gfCNCPoint5[21611] = {X 416.6146, Y 101.9777, Z -7.1667, A 0.000, B 0.000, C 0.000 }
gfCNCPoint5[21612] = {X 415.7067, Y 102.0800, Z -7.1667, A 0.000, B 0.000, C 0.000 }
gfCNCPoint5[21613] = {X 396.4059, Y 102.0800, Z -7.1667, A 0.000, B 0.000, C 0.000 }
gfCNCPoint5[21614] = {X 395.4981, Y 101.9777, Z -7.1667, A 0.000, B 0.000, C 0.000 }
gfCNCPoint5[21615] = {X 394.6357, Y 101.6760, Z -7.1667, A 0.000, B 0.000, C 0.000 }
gfCNCPoint5[21616] = {X 393.8621, Y 101.1899, Z -7.1667, A 0.000, B 0.000, C 0.000 }
gfCNCPoint5[21617] = {X 393.2161, Y 100.5438, Z -7.1667, A 0.000, B 0.000, C 0.000 }
gfCNCPoint5[21618] = {X 392.7300, Y 99.7702, Z -7.1667, A 0.000, B 0.000, C 0.000 }
gfCNCPoint5[21619] = {X 392.4282, Y 98.9079, Z -7.1667, A 0.000, B 0.000, C 0.000 }
gfCNCPoint5[21620] = {X 392.3259, Y 98.0000, Z -7.1667, A 0.000, B 0.000, C 0.000 }
gfCNCPoint5[21621] = {X 392.3259, Y 97.0659, Z -7.1667, A 0.000, B 0.000, C 0.000 }
gfCNCPoint5[21622] = {X 392.4280, Y 96.1590, Z -7.1667, A 0.000, B 0.000, C 0.000 }
gfCNCPoint5[21623] = {X 392.7292, Y 95.2974, Z -7.1667, A 0.000, B 0.000, C 0.000 }
gfCNCPoint5[21624] = {X 393.2143, Y 94.5244, Z -7.1667, A 0.000, B 0.000, C 0.000 }
gfCNCPoint5[21625] = {X 393.8591, Y 93.8785, Z -7.1667, A 0.000, B 0.000, C 0.000 }
gfCNCPoint5[21626] = {X 394.6313, Y 93.3921, Z -7.1667, A 0.000, B 0.000, C 0.000 }
gfCNCPoint5[21627] = {X 395.4924, Y 93.0895, Z -7.1667, A 0.000, B 0.000, C 0.000 }
gfCNCPoint5[21628] = {X 396.3991, Y 92.9859, Z -7.1667, A 0.000, B 0.000, C 0.000 }
gfCNCPoint5[21629] = {X 397.3627, Y 92.9425, Z -7.1667, A 0.000, B 0.000, C 0.000 }
gfCNCPoint5[21630] = {X 398.3229, Y 92.8515, Z -7.1667, A 0.000, B 0.000, C 0.000 }
gfCNCPoint5[21631] = {X 399.0264, Y 92.6809, Z -7.1667, A 0.000, B 0.000, C 0.000 }
gfCNCPoint5[21632] = {X 399.6742, Y 92.3580, Z -7.1667, A 0.000, B 0.000, C 0.000 }
gfCNCPoint5[21633] = {X 413.9281, Y 83.2302, Z -7.1667, A 0.000, B 0.000, C 0.000 }
gfCNCPoint5[21634] = {X 411.7658, Y 79.8536, Z -7.1667, A 0.000, B 0.000, C 0.000 }
gfCNCPoint5[21635] = {X 411.7676, Y 79.8524, Z -7.1667, A 0.000, B 0.000, C 0.000 }
gfCNCPoint5[21636] = {X 413.9660, Y 83.2895, Z -7.1667, A 0.000, B 0.000, C 0.000 }
gfCNCPoint5[21637] = {X 428.7544, Y 73.8309, Z -7.1667, A 0.000, B 0.000, C 0.000 }
gfCNCPoint5[21638] = {X 403.8726, Y 64.0690, Z -7.1667, A 0.000, B 0.000, C 0.000 }
gfCNCPoint5[21639] = {X 402.1412, Y 63.4961, Z -7.1667, A 0.000, B 0.000, C 0.000 }
gfCNCPoint5[21640] = {X 400.3574, Y 63.1162, Z -7.1667, A 0.000, B 0.000, C 0.000 }
gfCNCPoint5[21641] = {X 398.5427, Y 62.9340, Z -7.1667, A 0.000, B 0.000, C 0.000 }
gfCNCPoint5[21642] = {X 397.6551, Y 62.8309, Z -7.1667, A 0.000, B 0.000, C 0.000 }
gfCNCPoint5[21643] = {X 396.8125, Y 62.5333, Z -7.1667, A 0.000, B 0.000, C 0.000 }
gfCNCPoint5[21644] = {X 396.0571, Y 62.0560, Z -7.1667, A 0.000, B 0.000, C 0.000 }
gfCNCPoint5[21645] = {X 395.4264, Y 61.4230, Z -7.1667, A 0.000, B 0.000, C 0.000 }
gfCNCPoint5[21646] = {X 394.9520, Y 60.6657, Z -7.1667, A 0.000, B 0.000, C 0.000 }
gfCNCPoint5[21647] = {X 394.6575, Y 59.8221, Z -7.1667, A 0.000, B 0.000, C 0.000 }
gfCNCPoint5[21648] = {X 394.5577, Y 58.9341, Z -7.1667, A 0.000, B 0.000, C 0.000 }
gfCNCPoint5[21649] = {X 394.5577, Y 58.0000, Z -7.1667, A 0.000, B 0.000, C 0.000 }
gfCNCPoint5[21650] = {X 394.6580, Y 57.1099, Z -7.1667, A 0.000, B 0.000, C 0.000 }
gfCNCPoint5[21651] = {X 394.9538, Y 56.2645, Z -7.1667, A 0.000, B 0.000, C 0.000 }
gfCNCPoint5[21652] = {X 395.4304, Y 55.5060, Z -7.1667, A 0.000, B 0.000, C 0.000 }
gfCNCPoint5[21653] = {X 396.0638, Y 54.8727, Z -7.1667, A 0.000, B 0.000, C 0.000 }
gfCNCPoint5[21654] = {X 396.8222, Y 54.3961, Z -7.1667, A 0.000, B 0.000, C 0.000 }
gfCNCPoint5[21655] = {X 397.6676, Y 54.1003, Z -7.1667, A 0.000, B 0.000, C 0.000 }
gfCNCPoint5[21656] = {X 398.5577, Y 54.0000, Z -7.1667, A 0.000, B 0.000, C 0.000 }
gfCNCPoint5[21657] = {X 419.4886, Y 54.0000, Z -7.1667, A 0.000, B 0.000, C 0.000 }
gfCNCPoint5[21658] = {X 420.3787, Y 54.1003, Z -7.1667, A 0.000, B 0.000, C 0.000 }
gfCNCPoint5[21659] = {X 421.2241, Y 54.3961, Z -7.1667, A 0.000, B 0.000, C 0.000 }
gfCNCPoint5[21660] = {X 421.9826, Y 54.8727, Z -7.1667, A 0.000, B 0.000, C 0.000 }
gfCNCPoint5[21661] = {X 422.6159, Y 55.5060, Z -7.1667, A 0.000, B 0.000, C 0.000 }
gfCNCPoint5[21662] = {X 423.0925, Y 56.2645, Z -7.1667, A 0.000, B 0.000, C 0.000 }
gfCNCPoint5[21663] = {X 423.3883, Y 57.1099, Z -7.1667, A 0.000, B 0.000, C 0.000 }
gfCNCPoint5[21664] = {X 423.4886, Y 58.0000, Z -7.1667, A 0.000, B 0.000, C 0.000 }
gfCNCPoint5[21665] = {X 423.4886, Y 58.4503, Z -7.1667, A 0.000, B 0.000, C 0.000 }
gfCNCPoint5[21666] = {X 429.4945, Y 60.7902, Z -7.1667, A 0.000, B 0.000, C 0.000 }
gfCNCPoint5[21667] = {X 458.1780, Y 72.1710, Z -7.1667, A 0.000, B 0.000, C 0.000 }
gfCNCPoint5[21668] = {X 458.1783, Y 63.0394, Z -7.1667, A 0.000, B 0.000, C 0.000 }
gfCNCPoint5[21669] = {X 458.1841, Y 62.9246, Z -7.1667, A 0.000, B 0.000, C 0.000 }
gfCNCPoint5[21670] = {X 458.0117, Y 62.9089, Z -7.1667, A 0.000, B 0.000, C 0.000 }
gfCNCPoint5[21671] = {X 457.8402, Y 62.8858, Z -7.1667, A 0.000, B 0.000, C 0.000 }
gfCNCPoint5[21672] = {X 456.9338, Y 62.6316, Z -7.1667, A 0.000, B 0.000, C 0.000 }
gfCNCPoint5[21673] = {X 456.1119, Y 62.1727, Z -7.1667, A 0.000, B 0.000, C 0.000 }
gfCNCPoint5[21674] = {X 455.4201, Y 61.5343, Z -7.1667, A 0.000, B 0.000, C 0.000 }
gfCNCPoint5[21675] = {X 454.8966, Y 60.7519, Z -7.1667, A 0.000, B 0.000, C 0.000 }
gfCNCPoint5[21676] = {X 454.5704, Y 59.8689, Z -7.1667, A 0.000, B 0.000, C 0.000 }
gfCNCPoint5[21677] = {X 454.4596, Y 58.9341, Z -7.1667, A 0.000, B 0.000, C 0.000 }
gfCNCPoint5[21678] = {X 454.4596, Y 58.0000, Z -7.1667, A 0.000, B 0.000, C 0.000 }
gfCNCPoint5[21679] = {X 454.5599, Y 57.1099, Z -7.1667, A 0.000, B 0.000, C 0.000 }
gfCNCPoint5[21680] = {X 454.8557, Y 56.2645, Z -7.1667, A 0.000, B 0.000, C 0.000 }
gfCNCPoint5[21681] = {X 455.3323, Y 55.5060, Z -7.1667, A 0.000, B 0.000, C 0.000 }
gfCNCPoint5[21682] = {X 455.9656, Y 54.8727, Z -7.1667, A 0.000, B 0.000, C 0.000 }
gfCNCPoint5[21683] = {X 456.7241, Y 54.3961, Z -7.1667, A 0.000, B 0.000, C 0.000 }
gfCNCPoint5[21684] = {X 457.5695, Y 54.1003, Z -7.1667, A 0.000, B 0.000, C 0.000 }
gfCNCPoint5[21685] = {X 458.4596, Y 54.0000, Z -7.1667, A 0.000, B 0.000, C 0.000 }
gfCNCPoint5[21686] = {X 475.0000, Y 54.0000, Z -7.1667, A 0.000, B 0.000, C 0.000 }
gfCNCPoint5[21687] = {X 475.8901, Y 54.1003, Z -7.1667, A 0.000, B 0.000, C 0.000 }
gfCNCPoint5[21688] = {X 476.7355, Y 54.3961, Z -7.1667, A 0.000, B 0.000, C 0.000 }
gfCNCPoint5[21689] = {X 477.4940, Y 54.8727, Z -7.1667, A 0.000, B 0.000, C 0.000 }
gfCNCPoint5[21690] = {X 478.1273, Y 55.5060, Z -7.1667, A 0.000, B 0.000, C 0.000 }
gfCNCPoint5[21691] = {X 478.6039, Y 56.2645, Z -7.1667, A 0.000, B 0.000, C 0.000 }
gfCNCPoint5[21692] = {X 478.8997, Y 57.1099, Z -7.1667, A 0.000, B 0.000, C 0.000 }
gfCNCPoint5[21693] = {X 479.0000, Y 58.0000, Z -7.1667, A 0.000, B 0.000, C 0.000 }
gfCNCPoint5[21694] = {X 478.9999, Y 58.9671, Z -7.1667, A 0.000, B 0.000, C 0.000 }
gfCNCPoint5[21695] = {X 478.8827, Y 59.8957, Z -7.1667, A 0.000, B 0.000, C 0.000 }
gfCNCPoint5[21696] = {X 478.5529, Y 60.7716, Z -7.1667, A 0.000, B 0.000, C 0.000 }
gfCNCPoint5[21697] = {X 478.0287, Y 61.5469, Z -7.1667, A 0.000, B 0.000, C 0.000 }
gfCNCPoint5[21698] = {X 477.3386, Y 62.1792, Z -7.1667, A 0.000, B 0.000, C 0.000 }
gfCNCPoint5[21699] = {X 476.5204, Y 62.6338, Z -7.1667, A 0.000, B 0.000, C 0.000 }
gfCNCPoint5[21700] = {X 475.6191, Y 62.8859, Z -7.1667, A 0.000, B 0.000, C 0.000 }
gfCNCPoint5[21701] = {X 475.4521, Y 62.9084, Z -7.1667, A 0.000, B 0.000, C 0.000 }
gfCNCPoint5[21702] = {X 475.2843, Y 62.9240, Z -7.1667, A 0.000, B 0.000, C 0.000 }
gfCNCPoint5[21703] = {X 475.2810, Y 63.2811, Z -7.1667, A 0.000, B 0.000, C 0.000 }
gfCNCPoint5[21704] = {X 475.2814, Y 93.0285, Z -7.1667, A 0.000, B 0.000, C 0.000 }
gfCNCPoint5[21705] = {X 475.7846, Y 93.1405, Z -7.1667, A 0.000, B 0.000, C 0.000 }
gfCNCPoint5[21706] = {X 476.2789, Y 93.2866, Z -7.1667, A 0.000, B 0.000, C 0.000 }
gfCNCPoint5[21707] = {X 477.0319, Y 93.6280, Z -7.1667, A 0.000, B 0.000, C 0.000 }
gfCNCPoint5[21708] = {X 477.6982, Y 94.1177, Z -7.1667, A 0.000, B 0.000, C 0.000 }
gfCNCPoint5[21709] = {X 478.2488, Y 94.7346, Z -7.1667, A 0.000, B 0.000, C 0.000 }
gfCNCPoint5[21710] = {X 478.6600, Y 95.4519, Z -7.1667, A 0.000, B 0.000, C 0.000 }
gfCNCPoint5[21711] = {X 478.9141, Y 96.2388, Z -7.1667, A 0.000, B 0.000, C 0.000 }
gfCNCPoint5[21712] = {X 479.0000, Y 97.0611, Z -7.1667, A 0.000, B 0.000, C 0.000 }
gfCNCPoint5[21713] = {X 479.0000, Y 98.0000, Z -7.1667, A 0.000, B 0.000, C 0.000 }
gfCNCPoint5[21714] = {X 478.8997, Y 98.8901, Z -7.1667, A 0.000, B 0.000, C 0.000 }
gfCNCPoint5[21715] = {X 478.6039, Y 99.7355, Z -7.1667, A 0.000, B 0.000, C 0.000 }
gfCNCPoint5[21716] = {X 478.1273, Y 100.4940, Z -7.1667, A 0.000, B 0.000, C 0.000 }
gfCNCPoint5[21717] = {X 477.4940, Y 101.1273, Z -7.1667, A 0.000, B 0.000, C 0.000 }
gfCNCPoint5[21718] = {X 476.7355, Y 101.6039, Z -7.1667, A 0.000, B 0.000, C 0.000 }
gfCNCPoint5[21719] = {X 475.8901, Y 101.8997, Z -7.1667, A 0.000, B 0.000, C 0.000 }
gfCNCPoint5[21720] = {X 475.0000, Y 102.0000, Z -7.1667, A 0.000, B 0.000, C 0.000 }
gfCNCPoint5[21721] = {X 458.4596, Y 102.0000, Z -7.1667, A 0.000, B 0.000, C 0.000 }
gfCNCPoint5[21722] = {X 457.5695, Y 101.8997, Z -7.1667, A 0.000, B 0.000, C 0.000 }
gfCNCPoint5[21723] = {X 456.7241, Y 101.6039, Z -7.1667, A 0.000, B 0.000, C 0.000 }
gfCNCPoint5[21724] = {X 455.9656, Y 101.1273, Z -7.1667, A 0.000, B 0.000, C 0.000 }
gfCNCPoint5[21725] = {X 455.3323, Y 100.4940, Z -7.1667, A 0.000, B 0.000, C 0.000 }
gfCNCPoint5[21726] = {X 454.8557, Y 99.7355, Z -7.1667, A 0.000, B 0.000, C 0.000 }
gfCNCPoint5[21727] = {X 454.5599, Y 98.8901, Z -7.1667, A 0.000, B 0.000, C 0.000 }
gfCNCPoint5[21728] = {X 454.4596, Y 98.0000, Z -7.1667, A 0.000, B 0.000, C 0.000 }
gfCNCPoint5[21729] = {X 454.4596, Y 97.0659, Z -7.1667, A 0.000, B 0.000, C 0.000 }
gfCNCPoint5[21730] = {X 454.5511, Y 96.2154, Z -7.1667, A 0.000, B 0.000, C 0.000 }
gfCNCPoint5[21731] = {X 454.8213, Y 95.4037, Z -7.1667, A 0.000, B 0.000, C 0.000 }
gfCNCPoint5[21732] = {X 455.2580, Y 94.6681, Z -7.1667, A 0.000, B 0.000, C 0.000 }
gfCNCPoint5[21733] = {X 455.8411, Y 94.0422, Z -7.1667, A 0.000, B 0.000, C 0.000 }
gfCNCPoint5[21734] = {X 456.5439, Y 93.5545, Z -7.1667, A 0.000, B 0.000, C 0.000 }
gfCNCPoint5[21735] = {X 457.3344, Y 93.2275, Z -7.1667, A 0.000, B 0.000, C 0.000 }
gfCNCPoint5[21736] = {X 458.1763, Y 93.0760, Z -7.1667, A 0.000, B 0.000, C 0.000 }
gfCNCPoint5[21737] = {X 458.1763, Y 85.3767, Z -7.1667, A 0.000, B 0.000, C 0.000 }
gfCNCPoint5[21738] = {X 445.0152, Y 80.2175, Z -7.1667, A 0.000, B 0.000, C 0.000 }
gfCNCPoint5[21739] = {X 444.8242, Y 80.1425, Z -7.1667, A 0.000, B 0.000, C 0.000 }
gfCNCPoint5[21740] = {X 419.7033, Y 96.4151, Z -7.1667, A 0.000, B 0.000, C 0.000 }
gfCNCPoint5[21741] = {X 419.7067, Y 97.0659, Z -7.1667, A 0.000, B 0.000, C 0.000 }
gfCNCPoint5[21742] = {X 419.7067, Y 98.0000, Z -7.1667, A 0.000, B 0.000, C 0.000 }
gfCNCPoint5[21743] = {X 419.6064, Y 98.8901, Z -7.1667, A 0.000, B 0.000, C 0.000 }
gfCNCPoint5[21744] = {X 419.3106, Y 99.7355, Z -7.1667, A 0.000, B 0.000, C 0.000 }
gfCNCPoint5[21745] = {X 418.8340, Y 100.4940, Z -7.1667, A 0.000, B 0.000, C 0.000 }
gfCNCPoint5[21746] = {X 418.2007, Y 101.1273, Z -7.1667, A 0.000, B 0.000, C 0.000 }
gfCNCPoint5[21747] = {X 417.4422, Y 101.6039, Z -7.1667, A 0.000, B 0.000, C 0.000 }
gfCNCPoint5[21748] = {X 416.5968, Y 101.8997, Z -7.1667, A 0.000, B 0.000, C 0.000 }
gfCNCPoint5[21749] = {X 415.7067, Y 102.0000, Z -7.1667, A 0.000, B 0.000, C 0.000 }
gfCNCPoint5[21750] = {X 396.4059, Y 102.0000, Z -7.1667, A 0.000, B 0.000, C 0.000 }
gfCNCPoint5[21751] = {X 395.5159, Y 101.8997, Z -7.1667, A 0.000, B 0.000, C 0.000 }
gfCNCPoint5[21752] = {X 394.6704, Y 101.6039, Z -7.1667, A 0.000, B 0.000, C 0.000 }
gfCNCPoint5[21753] = {X 393.9120, Y 101.1273, Z -7.1667, A 0.000, B 0.000, C 0.000 }
gfCNCPoint5[21754] = {X 393.2786, Y 100.4940, Z -7.1667, A 0.000, B 0.000, C 0.000 }
gfCNCPoint5[21755] = {X 392.8021, Y 99.7355, Z -7.1667, A 0.000, B 0.000, C 0.000 }
gfCNCPoint5[21756] = {X 392.5062, Y 98.8901, Z -7.1667, A 0.000, B 0.000, C 0.000 }
gfCNCPoint5[21757] = {X 392.4059, Y 98.0000, Z -7.1667, A 0.000, B 0.000, C 0.000 }
gfCNCPoint5[21758] = {X 392.4059, Y 97.0659, Z -7.1667, A 0.000, B 0.000, C 0.000 }
gfCNCPoint5[21759] = {X 392.5060, Y 96.1767, Z -7.1667, A 0.000, B 0.000, C 0.000 }
gfCNCPoint5[21760] = {X 392.8013, Y 95.3319, Z -7.1667, A 0.000, B 0.000, C 0.000 }
gfCNCPoint5[21761] = {X 393.2770, Y 94.5740, Z -7.1667, A 0.000, B 0.000, C 0.000 }
gfCNCPoint5[21762] = {X 393.9093, Y 93.9407, Z -7.1667, A 0.000, B 0.000, C 0.000 }
gfCNCPoint5[21763] = {X 394.6666, Y 93.4639, Z -7.1667, A 0.000, B 0.000, C 0.000 }
gfCNCPoint5[21764] = {X 395.5109, Y 93.1674, Z -7.1667, A 0.000, B 0.000, C 0.000 }
gfCNCPoint5[21765] = {X 396.4000, Y 93.0659, Z -7.1667, A 0.000, B 0.000, C 0.000 }
gfCNCPoint5[21766] = {X 397.3680, Y 93.0223, Z -7.1667, A 0.000, B 0.000, C 0.000 }
gfCNCPoint5[21767] = {X 398.3327, Y 92.9309, Z -7.1667, A 0.000, B 0.000, C 0.000 }
gfCNCPoint5[21768] = {X 399.0537, Y 92.7561, Z -7.1667, A 0.000, B 0.000, C 0.000 }
gfCNCPoint5[21769] = {X 399.7177, Y 92.4252, Z -7.1667, A 0.000, B 0.000, C 0.000 }
gfCNCPoint5[21770] = {X 404.3153, Y 89.4621, Z -7.1667, A 0.000, B 0.000, C 0.000 }
gfCNCPoint5[21771] = {X 413.9660, Y 83.2895, Z -7.1667, A 0.000, B 0.000, C 0.000 }
gfCNCPoint5[21772] = {X 411.7676, Y 79.8524, Z -7.1667, A 0.000, B 0.000, C 0.000 }
gfCNCPoint5[21773] = {X 411.7676, Y 79.8524, Z -4.1667, A 0.000, B 0.000, C 0.000 }
gfCNCPoint5[21774] = {X 411.7676, Y 79.8524, Z 11.0000, A 0.000, B 0.000, C 0.000 }
gfCNCPoint5[21775] = {X 466.3117, Y 28.5934, Z 11.0000, A 0.000, B 0.000, C 0.000 }
gfCNCPoint5[21776] = {X 466.3117, Y 28.5934, Z -4.1667, A 0.000, B 0.000, C 0.000 }
gfCNCPoint5[21777] = {X 466.3117, Y 28.5934, Z -7.1667, A 0.000, B 0.000, C 0.000 }
gfCNCPoint5[21778] = {X 462.2317, Y 28.5935, Z -7.1667, A 0.000, B 0.000, C 0.000 }
gfCNCPoint5[21779] = {X 462.2320, Y 40.9142, Z -7.1667, A 0.000, B 0.000, C 0.000 }
gfCNCPoint5[21780] = {X 462.2403, Y 40.9211, Z -7.1667, A 0.000, B 0.000, C 0.000 }
gfCNCPoint5[21781] = {X 462.8748, Y 41.5915, Z -7.1667, A 0.000, B 0.000, C 0.000 }
gfCNCPoint5[21782] = {X 463.3524, Y 42.3815, Z -7.1667, A 0.000, B 0.000, C 0.000 }
gfCNCPoint5[21783] = {X 463.6513, Y 43.2548, Z -7.1667, A 0.000, B 0.000, C 0.000 }
gfCNCPoint5[21784] = {X 463.7578, Y 44.1718, Z -7.1667, A 0.000, B 0.000, C 0.000 }
gfCNCPoint5[21785] = {X 463.7579, Y 45.0000, Z -7.1667, A 0.000, B 0.000, C 0.000 }
gfCNCPoint5[21786] = {X 463.6496, Y 45.9613, Z -7.1667, A 0.000, B 0.000, C 0.000 }
gfCNCPoint5[21787] = {X 463.3301, Y 46.8744, Z -7.1667, A 0.000, B 0.000, C 0.000 }
gfCNCPoint5[21788] = {X 462.8155, Y 47.6935, Z -7.1667, A 0.000, B 0.000, C 0.000 }
gfCNCPoint5[21789] = {X 462.1314, Y 48.3775, Z -7.1667, A 0.000, B 0.000, C 0.000 }
gfCNCPoint5[21790] = {X 461.3123, Y 48.8922, Z -7.1667, A 0.000, B 0.000, C 0.000 }
gfCNCPoint5[21791] = {X 460.3992, Y 49.2117, Z -7.1667, A 0.000, B 0.000, C 0.000 }
gfCNCPoint5[21792] = {X 459.4379, Y 49.3200, Z -7.1667, A 0.000, B 0.000, C 0.000 }
gfCNCPoint5[21793] = {X 452.9945, Y 49.3200, Z -7.1667, A 0.000, B 0.000, C 0.000 }
gfCNCPoint5[21794] = {X 452.0380, Y 49.2128, Z -7.1667, A 0.000, B 0.000, C 0.000 }
gfCNCPoint5[21795] = {X 451.1291, Y 48.8965, Z -7.1667, A 0.000, B 0.000, C 0.000 }
gfCNCPoint5[21796] = {X 450.3127, Y 48.3868, Z -7.1667, A 0.000, B 0.000, C 0.000 }
gfCNCPoint5[21797] = {X 449.6294, Y 47.7091, Z -7.1667, A 0.000, B 0.000, C 0.000 }
gfCNCPoint5[21798] = {X 449.1132, Y 46.8968, Z -7.1667, A 0.000, B 0.000, C 0.000 }
gfCNCPoint5[21799] = {X 448.7895, Y 45.9905, Z -7.1667, A 0.000, B 0.000, C 0.000 }
gfCNCPoint5[21800] = {X 448.6746, Y 45.0349, Z -7.1667, A 0.000, B 0.000, C 0.000 }
gfCNCPoint5[21801] = {X 448.6749, Y 44.1494, Z -7.1667, A 0.000, B 0.000, C 0.000 }
gfCNCPoint5[21802] = {X 448.7853, Y 43.2364, Z -7.1667, A 0.000, B 0.000, C 0.000 }
gfCNCPoint5[21803] = {X 449.0865, Y 42.3675, Z -7.1667, A 0.000, B 0.000, C 0.000 }
gfCNCPoint5[21804] = {X 449.5648, Y 41.5821, Z -7.1667, A 0.000, B 0.000, C 0.000 }
gfCNCPoint5[21805] = {X 450.1984, Y 40.9157, Z -7.1667, A 0.000, B 0.000, C 0.000 }
gfCNCPoint5[21806] = {X 450.1984, Y 34.4738, Z -7.1667, A 0.000, B 0.000, C 0.000 }
gfCNCPoint5[21807] = {X 447.4755, Y 34.4738, Z -7.1667, A 0.000, B 0.000, C 0.000 }
gfCNCPoint5[21808] = {X 443.1901, Y 42.8178, Z -7.1667, A 0.000, B 0.000, C 0.000 }
gfCNCPoint5[21809] = {X 443.1949, Y 42.8312, Z -7.1667, A 0.000, B 0.000, C 0.000 }
gfCNCPoint5[21810] = {X 443.3606, Y 43.4918, Z -7.1667, A 0.000, B 0.000, C 0.000 }
gfCNCPoint5[21811] = {X 443.4203, Y 44.1703, Z -7.1667, A 0.000, B 0.000, C 0.000 }
gfCNCPoint5[21812] = {X 443.4205, Y 45.0000, Z -7.1667, A 0.000, B 0.000, C 0.000 }
gfCNCPoint5[21813] = {X 443.3122, Y 45.9613, Z -7.1667, A 0.000, B 0.000, C 0.000 }
gfCNCPoint5[21814] = {X 442.9927, Y 46.8744, Z -7.1667, A 0.000, B 0.000, C 0.000 }
gfCNCPoint5[21815] = {X 442.4780, Y 47.6935, Z -7.1667, A 0.000, B 0.000, C 0.000 }
gfCNCPoint5[21816] = {X 441.7939, Y 48.3775, Z -7.1667, A 0.000, B 0.000, C 0.000 }
gfCNCPoint5[21817] = {X 440.9748, Y 48.8922, Z -7.1667, A 0.000, B 0.000, C 0.000 }
gfCNCPoint5[21818] = {X 440.0618, Y 49.2117, Z -7.1667, A 0.000, B 0.000, C 0.000 }
gfCNCPoint5[21819] = {X 439.1005, Y 49.3200, Z -7.1667, A 0.000, B 0.000, C 0.000 }
gfCNCPoint5[21820] = {X 432.5144, Y 49.3200, Z -7.1667, A 0.000, B 0.000, C 0.000 }
gfCNCPoint5[21821] = {X 431.5531, Y 49.2117, Z -7.1667, A 0.000, B 0.000, C 0.000 }
gfCNCPoint5[21822] = {X 430.6401, Y 48.8922, Z -7.1667, A 0.000, B 0.000, C 0.000 }
gfCNCPoint5[21823] = {X 429.8210, Y 48.3775, Z -7.1667, A 0.000, B 0.000, C 0.000 }
gfCNCPoint5[21824] = {X 429.1369, Y 47.6935, Z -7.1667, A 0.000, B 0.000, C 0.000 }
gfCNCPoint5[21825] = {X 428.6223, Y 46.8745, Z -7.1667, A 0.000, B 0.000, C 0.000 }
gfCNCPoint5[21826] = {X 428.3027, Y 45.9614, Z -7.1667, A 0.000, B 0.000, C 0.000 }
gfCNCPoint5[21827] = {X 428.1944, Y 45.0001, Z -7.1667, A 0.000, B 0.000, C 0.000 }
gfCNCPoint5[21828] = {X 428.1948, Y 44.1494, Z -7.1667, A 0.000, B 0.000, C 0.000 }
gfCNCPoint5[21829] = {X 428.2925, Y 43.2935, Z -7.1667, A 0.000, B 0.000, C 0.000 }
gfCNCPoint5[21830] = {X 428.5580, Y 42.4740, Z -7.1667, A 0.000, B 0.000, C 0.000 }
gfCNCPoint5[21831] = {X 428.9809, Y 41.7236, Z -7.1667, A 0.000, B 0.000, C 0.000 }
gfCNCPoint5[21832] = {X 429.5442, Y 41.0719, Z -7.1667, A 0.000, B 0.000, C 0.000 }
gfCNCPoint5[21833] = {X 430.2256, Y 40.5449, Z -7.1667, A 0.000, B 0.000, C 0.000 }
gfCNCPoint5[21834] = {X 430.9981, Y 40.1637, Z -7.1667, A 0.000, B 0.000, C 0.000 }
gfCNCPoint5[21835] = {X 434.9867, Y 32.3563, Z -7.1667, A 0.000, B 0.000, C 0.000 }
gfCNCPoint5[21836] = {X 433.8226, Y 31.5747, Z -7.1667, A 0.000, B 0.000, C 0.000 }
gfCNCPoint5[21837] = {X 432.7640, Y 30.6552, Z -7.1667, A 0.000, B 0.000, C 0.000 }
gfCNCPoint5[21838] = {X 431.8273, Y 29.6119, Z -7.1667, A 0.000, B 0.000, C 0.000 }
gfCNCPoint5[21839] = {X 431.0267, Y 28.4607, Z -7.1667, A 0.000, B 0.000, C 0.000 }
gfCNCPoint5[21840] = {X 430.3746, Y 27.2194, Z -7.1667, A 0.000, B 0.000, C 0.000 }
gfCNCPoint5[21841] = {X 429.8811, Y 25.9069, Z -7.1667, A 0.000, B 0.000, C 0.000 }
gfCNCPoint5[21842] = {X 429.4497, Y 24.0606, Z -7.1667, A 0.000, B 0.000, C 0.000 }
gfCNCPoint5[21843] = {X 429.2325, Y 22.1770, Z -7.1667, A 0.000, B 0.000, C 0.000 }
gfCNCPoint5[21844] = {X 429.2323, Y 20.2810, Z -7.1667, A 0.000, B 0.000, C 0.000 }
gfCNCPoint5[21845] = {X 429.4491, Y 18.3974, Z -7.1667, A 0.000, B 0.000, C 0.000 }
gfCNCPoint5[21846] = {X 429.8800, Y 16.5509, Z -7.1667, A 0.000, B 0.000, C 0.000 }
gfCNCPoint5[21847] = {X 430.4498, Y 15.0197, Z -7.1667, A 0.000, B 0.000, C 0.000 }
gfCNCPoint5[21848] = {X 431.2251, Y 13.5816, Z -7.1667, A 0.000, B 0.000, C 0.000 }
gfCNCPoint5[21849] = {X 432.1911, Y 12.2641, Z -7.1667, A 0.000, B 0.000, C 0.000 }
gfCNCPoint5[21850] = {X 433.3295, Y 11.0922, Z -7.1667, A 0.000, B 0.000, C 0.000 }
gfCNCPoint5[21851] = {X 434.6185, Y 10.0883, Z -7.1667, A 0.000, B 0.000, C 0.000 }
gfCNCPoint5[21852] = {X 436.0334, Y 9.2716, Z -7.1667, A 0.000, B 0.000, C 0.000 }
gfCNCPoint5[21853] = {X 437.5474, Y 8.6577, Z -7.1667, A 0.000, B 0.000, C 0.000 }
gfCNCPoint5[21854] = {X 439.1316, Y 8.2581, Z -7.1667, A 0.000, B 0.000, C 0.000 }
gfCNCPoint5[21855] = {X 441.2286, Y 7.9678, Z -7.1667, A 0.000, B 0.000, C 0.000 }
gfCNCPoint5[21856] = {X 443.3436, Y 7.8736, Z -7.1667, A 0.000, B 0.000, C 0.000 }
gfCNCPoint5[21857] = {X 444.0357, Y 7.8696, Z -7.1667, A 0.000, B 0.000, C 0.000 }
gfCNCPoint5[21858] = {X 459.4469, Y 7.8696, Z -7.1667, A 0.000, B 0.000, C 0.000 }
gfCNCPoint5[21859] = {X 460.4062, Y 7.9777, Z -7.1667, A 0.000, B 0.000, C 0.000 }
gfCNCPoint5[21860] = {X 461.3174, Y 8.2965, Z -7.1667, A 0.000, B 0.000, C 0.000 }
gfCNCPoint5[21861] = {X 462.1348, Y 8.8101, Z -7.1667, A 0.000, B 0.000, C 0.000 }
gfCNCPoint5[21862] = {X 462.8174, Y 9.4927, Z -7.1667, A 0.000, B 0.000, C 0.000 }
gfCNCPoint5[21863] = {X 463.3310, Y 10.3101, Z -7.1667, A 0.000, B 0.000, C 0.000 }
gfCNCPoint5[21864] = {X 463.6499, Y 11.2213, Z -7.1667, A 0.000, B 0.000, C 0.000 }
gfCNCPoint5[21865] = {X 463.7579, Y 12.1806, Z -7.1667, A 0.000, B 0.000, C 0.000 }
gfCNCPoint5[21866] = {X 463.7579, Y 12.9782, Z -7.1667, A 0.000, B 0.000, C 0.000 }
gfCNCPoint5[21867] = {X 463.6566, Y 13.9077, Z -7.1667, A 0.000, B 0.000, C 0.000 }
gfCNCPoint5[21868] = {X 463.3577, Y 14.7936, Z -7.1667, A 0.000, B 0.000, C 0.000 }
gfCNCPoint5[21869] = {X 462.8751, Y 15.5945, Z -7.1667, A 0.000, B 0.000, C 0.000 }
gfCNCPoint5[21870] = {X 462.2315, Y 16.2728, Z -7.1667, A 0.000, B 0.000, C 0.000 }
gfCNCPoint5[21871] = {X 462.2317, Y 28.5935, Z -7.1667, A 0.000, B 0.000, C 0.000 }
gfCNCPoint5[21872] = {X 466.2317, Y 28.5934, Z -7.1667, A 0.000, B 0.000, C 0.000 }
gfCNCPoint5[21873] = {X 462.1517, Y 28.5935, Z -7.1667, A 0.000, B 0.000, C 0.000 }
gfCNCPoint5[21874] = {X 462.1520, Y 40.9519, Z -7.1667, A 0.000, B 0.000, C 0.000 }
gfCNCPoint5[21875] = {X 462.1889, Y 40.9824, Z -7.1667, A 0.000, B 0.000, C 0.000 }
gfCNCPoint5[21876] = {X 462.8115, Y 41.6404, Z -7.1667, A 0.000, B 0.000, C 0.000 }
gfCNCPoint5[21877] = {X 463.2801, Y 42.4156, Z -7.1667, A 0.000, B 0.000, C 0.000 }
gfCNCPoint5[21878] = {X 463.5733, Y 43.2726, Z -7.1667, A 0.000, B 0.000, C 0.000 }
gfCNCPoint5[21879] = {X 463.6778, Y 44.1724, Z -7.1667, A 0.000, B 0.000, C 0.000 }
gfCNCPoint5[21880] = {X 463.6779, Y 45.0000, Z -7.1667, A 0.000, B 0.000, C 0.000 }
gfCNCPoint5[21881] = {X 463.5716, Y 45.9435, Z -7.1667, A 0.000, B 0.000, C 0.000 }
gfCNCPoint5[21882] = {X 463.2580, Y 46.8397, Z -7.1667, A 0.000, B 0.000, C 0.000 }
gfCNCPoint5[21883] = {X 462.7529, Y 47.6436, Z -7.1667, A 0.000, B 0.000, C 0.000 }
gfCNCPoint5[21884] = {X 462.0815, Y 48.3150, Z -7.1667, A 0.000, B 0.000, C 0.000 }
gfCNCPoint5[21885] = {X 461.2776, Y 48.8201, Z -7.1667, A 0.000, B 0.000, C 0.000 }
gfCNCPoint5[21886] = {X 460.3814, Y 49.1337, Z -7.1667, A 0.000, B 0.000, C 0.000 }
gfCNCPoint5[21887] = {X 459.4379, Y 49.2400, Z -7.1667, A 0.000, B 0.000, C 0.000 }
gfCNCPoint5[21888] = {X 452.9945, Y 49.2400, Z -7.1667, A 0.000, B 0.000, C 0.000 }
gfCNCPoint5[21889] = {X 452.0558, Y 49.1348, Z -7.1667, A 0.000, B 0.000, C 0.000 }
gfCNCPoint5[21890] = {X 451.1636, Y 48.8243, Z -7.1667, A 0.000, B 0.000, C 0.000 }
gfCNCPoint5[21891] = {X 450.3624, Y 48.3241, Z -7.1667, A 0.000, B 0.000, C 0.000 }
gfCNCPoint5[21892] = {X 449.6918, Y 47.6589, Z -7.1667, A 0.000, B 0.000, C 0.000 }
gfCNCPoint5[21893] = {X 449.1851, Y 46.8617, Z -7.1667, A 0.000, B 0.000, C 0.000 }
gfCNCPoint5[21894] = {X 448.8674, Y 45.9721, Z -7.1667, A 0.000, B 0.000, C 0.000 }
gfCNCPoint5[21895] = {X 448.7546, Y 45.0343, Z -7.1667, A 0.000, B 0.000, C 0.000 }
gfCNCPoint5[21896] = {X 448.7549, Y 44.1505, Z -7.1667, A 0.000, B 0.000, C 0.000 }
gfCNCPoint5[21897] = {X 448.8654, Y 43.2454, Z -7.1667, A 0.000, B 0.000, C 0.000 }
gfCNCPoint5[21898] = {X 449.1668, Y 42.3850, Z -7.1667, A 0.000, B 0.000, C 0.000 }
gfCNCPoint5[21899] = {X 449.6452, Y 41.6088, Z -7.1667, A 0.000, B 0.000, C 0.000 }
gfCNCPoint5[21900] = {X 450.2784, Y 40.9529, Z -7.1667, A 0.000, B 0.000, C 0.000 }
gfCNCPoint5[21901] = {X 450.2784, Y 34.3938, Z -7.1667, A 0.000, B 0.000, C 0.000 }
gfCNCPoint5[21902] = {X 447.4266, Y 34.3938, Z -7.1667, A 0.000, B 0.000, C 0.000 }
gfCNCPoint5[21903] = {X 443.1031, Y 42.8122, Z -7.1667, A 0.000, B 0.000, C 0.000 }
gfCNCPoint5[21904] = {X 443.1194, Y 42.8575, Z -7.1667, A 0.000, B 0.000, C 0.000 }
gfCNCPoint5[21905] = {X 443.2817, Y 43.5055, Z -7.1667, A 0.000, B 0.000, C 0.000 }
gfCNCPoint5[21906] = {X 443.3403, Y 44.1710, Z -7.1667, A 0.000, B 0.000, C 0.000 }
gfCNCPoint5[21907] = {X 443.3405, Y 45.0000, Z -7.1667, A 0.000, B 0.000, C 0.000 }
gfCNCPoint5[21908] = {X 443.2342, Y 45.9435, Z -7.1667, A 0.000, B 0.000, C 0.000 }
gfCNCPoint5[21909] = {X 442.9206, Y 46.8397, Z -7.1667, A 0.000, B 0.000, C 0.000 }
gfCNCPoint5[21910] = {X 442.4154, Y 47.6436, Z -7.1667, A 0.000, B 0.000, C 0.000 }
gfCNCPoint5[21911] = {X 441.7441, Y 48.3150, Z -7.1667, A 0.000, B 0.000, C 0.000 }
gfCNCPoint5[21912] = {X 440.9401, Y 48.8201, Z -7.1667, A 0.000, B 0.000, C 0.000 }
gfCNCPoint5[21913] = {X 440.0440, Y 49.1337, Z -7.1667, A 0.000, B 0.000, C 0.000 }
gfCNCPoint5[21914] = {X 439.1005, Y 49.2400, Z -7.1667, A 0.000, B 0.000, C 0.000 }
gfCNCPoint5[21915] = {X 432.5144, Y 49.2400, Z -7.1667, A 0.000, B 0.000, C 0.000 }
gfCNCPoint5[21916] = {X 431.5709, Y 49.1337, Z -7.1667, A 0.000, B 0.000, C 0.000 }
gfCNCPoint5[21917] = {X 430.6748, Y 48.8201, Z -7.1667, A 0.000, B 0.000, C 0.000 }
gfCNCPoint5[21918] = {X 429.8708, Y 48.3150, Z -7.1667, A 0.000, B 0.000, C 0.000 }
gfCNCPoint5[21919] = {X 429.1995, Y 47.6436, Z -7.1667, A 0.000, B 0.000, C 0.000 }
gfCNCPoint5[21920] = {X 428.6943, Y 46.8397, Z -7.1667, A 0.000, B 0.000, C 0.000 }
gfCNCPoint5[21921] = {X 428.3807, Y 45.9436, Z -7.1667, A 0.000, B 0.000, C 0.000 }
gfCNCPoint5[21922] = {X 428.2744, Y 45.0001, Z -7.1667, A 0.000, B 0.000, C 0.000 }
gfCNCPoint5[21923] = {X 428.2748, Y 44.1505, Z -7.1667, A 0.000, B 0.000, C 0.000 }
gfCNCPoint5[21924] = {X 428.3718, Y 43.3054, Z -7.1667, A 0.000, B 0.000, C 0.000 }
gfCNCPoint5[21925] = {X 428.6354, Y 42.4967, Z -7.1667, A 0.000, B 0.000, C 0.000 }
gfCNCPoint5[21926] = {X 429.0552, Y 41.7570, Z -7.1667, A 0.000, B 0.000, C 0.000 }
gfCNCPoint5[21927] = {X 429.6142, Y 41.1158, Z -7.1667, A 0.000, B 0.000, C 0.000 }
gfCNCPoint5[21928] = {X 430.2899, Y 40.5992, Z -7.1667, A 0.000, B 0.000, C 0.000 }
gfCNCPoint5[21929] = {X 431.0551, Y 40.2278, Z -7.1667, A 0.000, B 0.000, C 0.000 }
gfCNCPoint5[21930] = {X 435.0924, Y 32.3252, Z -7.1667, A 0.000, B 0.000, C 0.000 }
gfCNCPoint5[21931] = {X 433.9213, Y 31.5493, Z -7.1667, A 0.000, B 0.000, C 0.000 }
gfCNCPoint5[21932] = {X 432.8561, Y 30.6334, Z -7.1667, A 0.000, B 0.000, C 0.000 }
gfCNCPoint5[21933] = {X 431.9135, Y 29.5918, Z -7.1667, A 0.000, B 0.000, C 0.000 }
gfCNCPoint5[21934] = {X 431.1082, Y 28.4407, Z -7.1667, A 0.000, B 0.000, C 0.000 }
gfCNCPoint5[21935] = {X 430.4528, Y 27.1981, Z -7.1667, A 0.000, B 0.000, C 0.000 }
gfCNCPoint5[21936] = {X 429.9575, Y 25.8835, Z -7.1667, A 0.000, B 0.000, C 0.000 }
gfCNCPoint5[21937] = {X 429.5284, Y 24.0462, Z -7.1667, A 0.000, B 0.000, C 0.000 }
gfCNCPoint5[21938] = {X 429.3124, Y 22.1719, Z -7.1667, A 0.000, B 0.000, C 0.000 }
gfCNCPoint5[21939] = {X 429.3122, Y 20.2852, Z -7.1667, A 0.000, B 0.000, C 0.000 }
gfCNCPoint5[21940] = {X 429.5280, Y 18.4109, Z -7.1667, A 0.000, B 0.000, C 0.000 }
gfCNCPoint5[21941] = {X 429.9568, Y 16.5735, Z -7.1667, A 0.000, B 0.000, C 0.000 }
gfCNCPoint5[21942] = {X 430.5227, Y 15.0527, Z -7.1667, A 0.000, B 0.000, C 0.000 }
gfCNCPoint5[21943] = {X 431.2928, Y 13.6243, Z -7.1667, A 0.000, B 0.000, C 0.000 }
gfCNCPoint5[21944] = {X 432.2523, Y 12.3156, Z -7.1667, A 0.000, B 0.000, C 0.000 }
gfCNCPoint5[21945] = {X 433.3830, Y 11.1517, Z -7.1667, A 0.000, B 0.000, C 0.000 }
gfCNCPoint5[21946] = {X 434.6633, Y 10.1546, Z -7.1667, A 0.000, B 0.000, C 0.000 }
gfCNCPoint5[21947] = {X 436.0687, Y 9.3434, Z -7.1667, A 0.000, B 0.000, C 0.000 }
gfCNCPoint5[21948] = {X 437.5726, Y 8.7336, Z -7.1667, A 0.000, B 0.000, C 0.000 }
gfCNCPoint5[21949] = {X 439.1460, Y 8.3368, Z -7.1667, A 0.000, B 0.000, C 0.000 }
gfCNCPoint5[21950] = {X 441.2360, Y 8.0474, Z -7.1667, A 0.000, B 0.000, C 0.000 }
gfCNCPoint5[21951] = {X 443.3437, Y 7.9536, Z -7.1667, A 0.000, B 0.000, C 0.000 }
gfCNCPoint5[21952] = {X 444.0360, Y 7.9496, Z -7.1667, A 0.000, B 0.000, C 0.000 }
gfCNCPoint5[21953] = {X 459.4469, Y 7.9496, Z -7.1667, A 0.000, B 0.000, C 0.000 }
gfCNCPoint5[21954] = {X 460.3884, Y 8.0556, Z -7.1667, A 0.000, B 0.000, C 0.000 }
gfCNCPoint5[21955] = {X 461.2827, Y 8.3686, Z -7.1667, A 0.000, B 0.000, C 0.000 }
gfCNCPoint5[21956] = {X 462.0849, Y 8.8727, Z -7.1667, A 0.000, B 0.000, C 0.000 }
gfCNCPoint5[21957] = {X 462.7549, Y 9.5426, Z -7.1667, A 0.000, B 0.000, C 0.000 }
gfCNCPoint5[21958] = {X 463.2589, Y 10.3448, Z -7.1667, A 0.000, B 0.000, C 0.000 }
gfCNCPoint5[21959] = {X 463.5719, Y 11.2391, Z -7.1667, A 0.000, B 0.000, C 0.000 }
gfCNCPoint5[21960] = {X 463.6779, Y 12.1806, Z -7.1667, A 0.000, B 0.000, C 0.000 }
gfCNCPoint5[21961] = {X 463.6779, Y 12.9782, Z -7.1667, A 0.000, B 0.000, C 0.000 }
gfCNCPoint5[21962] = {X 463.5765, Y 13.8995, Z -7.1667, A 0.000, B 0.000, C 0.000 }
gfCNCPoint5[21963] = {X 463.2773, Y 14.7767, Z -7.1667, A 0.000, B 0.000, C 0.000 }
gfCNCPoint5[21964] = {X 462.7946, Y 15.5680, Z -7.1667, A 0.000, B 0.000, C 0.000 }
gfCNCPoint5[21965] = {X 462.1515, Y 16.2355, Z -7.1667, A 0.000, B 0.000, C 0.000 }
gfCNCPoint5[21966] = {X 462.1517, Y 28.5935, Z -7.1667, A 0.000, B 0.000, C 0.000 }
gfCNCPoint5[21967] = {X 466.1517, Y 28.5934, Z -7.1667, A 0.000, B 0.000, C 0.000 }
gfCNCPoint5[21968] = {X 462.0717, Y 28.5935, Z -7.1667, A 0.000, B 0.000, C 0.000 }
gfCNCPoint5[21969] = {X 462.0720, Y 40.9895, Z -7.1667, A 0.000, B 0.000, C 0.000 }
gfCNCPoint5[21970] = {X 462.1375, Y 41.0436, Z -7.1667, A 0.000, B 0.000, C 0.000 }
gfCNCPoint5[21971] = {X 462.7481, Y 41.6892, Z -7.1667, A 0.000, B 0.000, C 0.000 }
gfCNCPoint5[21972] = {X 463.2077, Y 42.4497, Z -7.1667, A 0.000, B 0.000, C 0.000 }
gfCNCPoint5[21973] = {X 463.4953, Y 43.2905, Z -7.1667, A 0.000, B 0.000, C 0.000 }
gfCNCPoint5[21974] = {X 463.5978, Y 44.1731, Z -7.1667, A 0.000, B 0.000, C 0.000 }
gfCNCPoint5[21975] = {X 463.5979, Y 45.0000, Z -7.1667, A 0.000, B 0.000, C 0.000 }
gfCNCPoint5[21976] = {X 463.4936, Y 45.9257, Z -7.1667, A 0.000, B 0.000, C 0.000 }
gfCNCPoint5[21977] = {X 463.1860, Y 46.8050, Z -7.1667, A 0.000, B 0.000, C 0.000 }
gfCNCPoint5[21978] = {X 462.6904, Y 47.5937, Z -7.1667, A 0.000, B 0.000, C 0.000 }
gfCNCPoint5[21979] = {X 462.0317, Y 48.2524, Z -7.1667, A 0.000, B 0.000, C 0.000 }
gfCNCPoint5[21980] = {X 461.2429, Y 48.7480, Z -7.1667, A 0.000, B 0.000, C 0.000 }
gfCNCPoint5[21981] = {X 460.3636, Y 49.0557, Z -7.1667, A 0.000, B 0.000, C 0.000 }
gfCNCPoint5[21982] = {X 459.4379, Y 49.1600, Z -7.1667, A 0.000, B 0.000, C 0.000 }
gfCNCPoint5[21983] = {X 452.9945, Y 49.1600, Z -7.1667, A 0.000, B 0.000, C 0.000 }
gfCNCPoint5[21984] = {X 452.0735, Y 49.0568, Z -7.1667, A 0.000, B 0.000, C 0.000 }
gfCNCPoint5[21985] = {X 451.1982, Y 48.7522, Z -7.1667, A 0.000, B 0.000, C 0.000 }
gfCNCPoint5[21986] = {X 450.4120, Y 48.2614, Z -7.1667, A 0.000, B 0.000, C 0.000 }
gfCNCPoint5[21987] = {X 449.7541, Y 47.6087, Z -7.1667, A 0.000, B 0.000, C 0.000 }
gfCNCPoint5[21988] = {X 449.2569, Y 46.8266, Z -7.1667, A 0.000, B 0.000, C 0.000 }
gfCNCPoint5[21989] = {X 448.9453, Y 45.9538, Z -7.1667, A 0.000, B 0.000, C 0.000 }
gfCNCPoint5[21990] = {X 448.8346, Y 45.0336, Z -7.1667, A 0.000, B 0.000, C 0.000 }
gfCNCPoint5[21991] = {X 448.8349, Y 44.1516, Z -7.1667, A 0.000, B 0.000, C 0.000 }
gfCNCPoint5[21992] = {X 448.9454, Y 43.2545, Z -7.1667, A 0.000, B 0.000, C 0.000 }
gfCNCPoint5[21993] = {X 449.2471, Y 42.4026, Z -7.1667, A 0.000, B 0.000, C 0.000 }
gfCNCPoint5[21994] = {X 449.7256, Y 41.6358, Z -7.1667, A 0.000, B 0.000, C 0.000 }
gfCNCPoint5[21995] = {X 450.3584, Y 40.9906, Z -7.1667, A 0.000, B 0.000, C 0.000 }
gfCNCPoint5[21996] = {X 450.3584, Y 34.3138, Z -7.1667, A 0.000, B 0.000, C 0.000 }
gfCNCPoint5[21997] = {X 447.3778, Y 34.3138, Z -7.1667, A 0.000, B 0.000, C 0.000 }
gfCNCPoint5[21998] = {X 443.0161, Y 42.8065, Z -7.1667, A 0.000, B 0.000, C 0.000 }
gfCNCPoint5[21999] = {X 443.0438, Y 42.8837, Z -7.1667, A 0.000, B 0.000, C 0.000 }
gfCNCPoint5[22000] = {X 443.2029, Y 43.5192, Z -7.1667, A 0.000, B 0.000, C 0.000 }
gfCNCPoint5[22001] = {X 443.2603, Y 44.1717, Z -7.1667, A 0.000, B 0.000, C 0.000 }
gfCNCPoint5[22002] = {X 443.2605, Y 45.0000, Z -7.1667, A 0.000, B 0.000, C 0.000 }
gfCNCPoint5[22003] = {X 443.1562, Y 45.9257, Z -7.1667, A 0.000, B 0.000, C 0.000 }
gfCNCPoint5[22004] = {X 442.8485, Y 46.8050, Z -7.1667, A 0.000, B 0.000, C 0.000 }
gfCNCPoint5[22005] = {X 442.3529, Y 47.5937, Z -7.1667, A 0.000, B 0.000, C 0.000 }
gfCNCPoint5[22006] = {X 441.6942, Y 48.2524, Z -7.1667, A 0.000, B 0.000, C 0.000 }
gfCNCPoint5[22007] = {X 440.9054, Y 48.7480, Z -7.1667, A 0.000, B 0.000, C 0.000 }
gfCNCPoint5[22008] = {X 440.0262, Y 49.0557, Z -7.1667, A 0.000, B 0.000, C 0.000 }
gfCNCPoint5[22009] = {X 439.1005, Y 49.1600, Z -7.1667, A 0.000, B 0.000, C 0.000 }
gfCNCPoint5[22010] = {X 432.5144, Y 49.1600, Z -7.1667, A 0.000, B 0.000, C 0.000 }
gfCNCPoint5[22011] = {X 431.5887, Y 49.0557, Z -7.1667, A 0.000, B 0.000, C 0.000 }
gfCNCPoint5[22012] = {X 430.7095, Y 48.7480, Z -7.1667, A 0.000, B 0.000, C 0.000 }
gfCNCPoint5[22013] = {X 429.9207, Y 48.2524, Z -7.1667, A 0.000, B 0.000, C 0.000 }
gfCNCPoint5[22014] = {X 429.2620, Y 47.5937, Z -7.1667, A 0.000, B 0.000, C 0.000 }
gfCNCPoint5[22015] = {X 428.7664, Y 46.8050, Z -7.1667, A 0.000, B 0.000, C 0.000 }
gfCNCPoint5[22016] = {X 428.4587, Y 45.9257, Z -7.1667, A 0.000, B 0.000, C 0.000 }
gfCNCPoint5[22017] = {X 428.3544, Y 45.0000, Z -7.1667, A 0.000, B 0.000, C 0.000 }
gfCNCPoint5[22018] = {X 428.3548, Y 44.1516, Z -7.1667, A 0.000, B 0.000, C 0.000 }
gfCNCPoint5[22019] = {X 428.4510, Y 43.3174, Z -7.1667, A 0.000, B 0.000, C 0.000 }
gfCNCPoint5[22020] = {X 428.7128, Y 42.5195, Z -7.1667, A 0.000, B 0.000, C 0.000 }
gfCNCPoint5[22021] = {X 429.1295, Y 41.7905, Z -7.1667, A 0.000, B 0.000, C 0.000 }
gfCNCPoint5[22022] = {X 429.6841, Y 41.1600, Z -7.1667, A 0.000, B 0.000, C 0.000 }
gfCNCPoint5[22023] = {X 430.3541, Y 40.6537, Z -7.1667, A 0.000, B 0.000, C 0.000 }
gfCNCPoint5[22024] = {X 431.1120, Y 40.2923, Z -7.1667, A 0.000, B 0.000, C 0.000 }
gfCNCPoint5[22025] = {X 435.1984, Y 32.2936, Z -7.1667, A 0.000, B 0.000, C 0.000 }
gfCNCPoint5[22026] = {X 434.0202, Y 31.5236, Z -7.1667, A 0.000, B 0.000, C 0.000 }
gfCNCPoint5[22027] = {X 432.9483, Y 30.6115, Z -7.1667, A 0.000, B 0.000, C 0.000 }
gfCNCPoint5[22028] = {X 431.9998, Y 29.5716, Z -7.1667, A 0.000, B 0.000, C 0.000 }
gfCNCPoint5[22029] = {X 431.1897, Y 28.4206, Z -7.1667, A 0.000, B 0.000, C 0.000 }
gfCNCPoint5[22030] = {X 430.5310, Y 27.1768, Z -7.1667, A 0.000, B 0.000, C 0.000 }
gfCNCPoint5[22031] = {X 430.0340, Y 25.8600, Z -7.1667, A 0.000, B 0.000, C 0.000 }
gfCNCPoint5[22032] = {X 429.6071, Y 24.0318, Z -7.1667, A 0.000, B 0.000, C 0.000 }
gfCNCPoint5[22033] = {X 429.3922, Y 22.1668, Z -7.1667, A 0.000, B 0.000, C 0.000 }
gfCNCPoint5[22034] = {X 429.3921, Y 20.2894, Z -7.1667, A 0.000, B 0.000, C 0.000 }
gfCNCPoint5[22035] = {X 429.6068, Y 18.4244, Z -7.1667, A 0.000, B 0.000, C 0.000 }
gfCNCPoint5[22036] = {X 430.0335, Y 16.5962, Z -7.1667, A 0.000, B 0.000, C 0.000 }
gfCNCPoint5[22037] = {X 430.5956, Y 15.0856, Z -7.1667, A 0.000, B 0.000, C 0.000 }
gfCNCPoint5[22038] = {X 431.3605, Y 13.6669, Z -7.1667, A 0.000, B 0.000, C 0.000 }
gfCNCPoint5[22039] = {X 432.3135, Y 12.3672, Z -7.1667, A 0.000, B 0.000, C 0.000 }
gfCNCPoint5[22040] = {X 433.4365, Y 11.2111, Z -7.1667, A 0.000, B 0.000, C 0.000 }
gfCNCPoint5[22041] = {X 434.7081, Y 10.2208, Z -7.1667, A 0.000, B 0.000, C 0.000 }
gfCNCPoint5[22042] = {X 436.1040, Y 9.4152, Z -7.1667, A 0.000, B 0.000, C 0.000 }
gfCNCPoint5[22043] = {X 437.5977, Y 8.8096, Z -7.1667, A 0.000, B 0.000, C 0.000 }
gfCNCPoint5[22044] = {X 439.1605, Y 8.4155, Z -7.1667, A 0.000, B 0.000, C 0.000 }
gfCNCPoint5[22045] = {X 441.2433, Y 8.1271, Z -7.1667, A 0.000, B 0.000, C 0.000 }
gfCNCPoint5[22046] = {X 443.3439, Y 8.0336, Z -7.1667, A 0.000, B 0.000, C 0.000 }
gfCNCPoint5[22047] = {X 444.0362, Y 8.0296, Z -7.1667, A 0.000, B 0.000, C 0.000 }
gfCNCPoint5[22048] = {X 459.4469, Y 8.0296, Z -7.1667, A 0.000, B 0.000, C 0.000 }
gfCNCPoint5[22049] = {X 460.3706, Y 8.1336, Z -7.1667, A 0.000, B 0.000, C 0.000 }
gfCNCPoint5[22050] = {X 461.2479, Y 8.4407, Z -7.1667, A 0.000, B 0.000, C 0.000 }
gfCNCPoint5[22051] = {X 462.0350, Y 8.9352, Z -7.1667, A 0.000, B 0.000, C 0.000 }
gfCNCPoint5[22052] = {X 462.6923, Y 9.5925, Z -7.1667, A 0.000, B 0.000, C 0.000 }
gfCNCPoint5[22053] = {X 463.1869, Y 10.3796, Z -7.1667, A 0.000, B 0.000, C 0.000 }
gfCNCPoint5[22054] = {X 463.4939, Y 11.2569, Z -7.1667, A 0.000, B 0.000, C 0.000 }
gfCNCPoint5[22055] = {X 463.5979, Y 12.1806, Z -7.1667, A 0.000, B 0.000, C 0.000 }
gfCNCPoint5[22056] = {X 463.5979, Y 12.9782, Z -7.1667, A 0.000, B 0.000, C 0.000 }
gfCNCPoint5[22057] = {X 463.5023, Y 13.8648, Z -7.1667, A 0.000, B 0.000, C 0.000 }
gfCNCPoint5[22058] = {X 463.2199, Y 14.7107, Z -7.1667, A 0.000, B 0.000, C 0.000 }
gfCNCPoint5[22059] = {X 462.7637, Y 15.4770, Z -7.1667, A 0.000, B 0.000, C 0.000 }
gfCNCPoint5[22060] = {X 462.1547, Y 16.1284, Z -7.1667, A 0.000, B 0.000, C 0.000 }
gfCNCPoint5[22061] = {X 462.0715, Y 16.1982, Z -7.1667, A 0.000, B 0.000, C 0.000 }
gfCNCPoint5[22062] = {X 462.0717, Y 28.5935, Z -7.1667, A 0.000, B 0.000, C 0.000 }
gfCNCPoint5[22063] = {X 466.0717, Y 28.5934, Z -7.1667, A 0.000, B 0.000, C 0.000 }
gfCNCPoint5[22064] = {X 461.9917, Y 28.5935, Z -7.1667, A 0.000, B 0.000, C 0.000 }
gfCNCPoint5[22065] = {X 461.9920, Y 41.0272, Z -7.1667, A 0.000, B 0.000, C 0.000 }
gfCNCPoint5[22066] = {X 462.0860, Y 41.1049, Z -7.1667, A 0.000, B 0.000, C 0.000 }
gfCNCPoint5[22067] = {X 462.6847, Y 41.7380, Z -7.1667, A 0.000, B 0.000, C 0.000 }
gfCNCPoint5[22068] = {X 463.1353, Y 42.4838, Z -7.1667, A 0.000, B 0.000, C 0.000 }
gfCNCPoint5[22069] = {X 463.4173, Y 43.3083, Z -7.1667, A 0.000, B 0.000, C 0.000 }
gfCNCPoint5[22070] = {X 463.5178, Y 44.1738, Z -7.1667, A 0.000, B 0.000, C 0.000 }
gfCNCPoint5[22071] = {X 463.5179, Y 45.0000, Z -7.1667, A 0.000, B 0.000, C 0.000 }
gfCNCPoint5[22072] = {X 463.4156, Y 45.9079, Z -7.1667, A 0.000, B 0.000, C 0.000 }
gfCNCPoint5[22073] = {X 463.1139, Y 46.7702, Z -7.1667, A 0.000, B 0.000, C 0.000 }
gfCNCPoint5[22074] = {X 462.6278, Y 47.5438, Z -7.1667, A 0.000, B 0.000, C 0.000 }
gfCNCPoint5[22075] = {X 461.9818, Y 48.1899, Z -7.1667, A 0.000, B 0.000, C 0.000 }
gfCNCPoint5[22076] = {X 461.2082, Y 48.6760, Z -7.1667, A 0.000, B 0.000, C 0.000 }
gfCNCPoint5[22077] = {X 460.3458, Y 48.9777, Z -7.1667, A 0.000, B 0.000, C 0.000 }
gfCNCPoint5[22078] = {X 459.4379, Y 49.0800, Z -7.1667, A 0.000, B 0.000, C 0.000 }
gfCNCPoint5[22079] = {X 452.9945, Y 49.0800, Z -7.1667, A 0.000, B 0.000, C 0.000 }
gfCNCPoint5[22080] = {X 452.0912, Y 48.9788, Z -7.1667, A 0.000, B 0.000, C 0.000 }
gfCNCPoint5[22081] = {X 451.2327, Y 48.6800, Z -7.1667, A 0.000, B 0.000, C 0.000 }
gfCNCPoint5[22082] = {X 450.4617, Y 48.1987, Z -7.1667, A 0.000, B 0.000, C 0.000 }
gfCNCPoint5[22083] = {X 449.8164, Y 47.5585, Z -7.1667, A 0.000, B 0.000, C 0.000 }
gfCNCPoint5[22084] = {X 449.3288, Y 46.7914, Z -7.1667, A 0.000, B 0.000, C 0.000 }
gfCNCPoint5[22085] = {X 449.0232, Y 45.9354, Z -7.1667, A 0.000, B 0.000, C 0.000 }
gfCNCPoint5[22086] = {X 448.9146, Y 45.0330, Z -7.1667, A 0.000, B 0.000, C 0.000 }
gfCNCPoint5[22087] = {X 448.9149, Y 44.1527, Z -7.1667, A 0.000, B 0.000, C 0.000 }
gfCNCPoint5[22088] = {X 449.0254, Y 43.2637, Z -7.1667, A 0.000, B 0.000, C 0.000 }
gfCNCPoint5[22089] = {X 449.3274, Y 42.4203, Z -7.1667, A 0.000, B 0.000, C 0.000 }
gfCNCPoint5[22090] = {X 449.8061, Y 41.6631, Z -7.1667, A 0.000, B 0.000, C 0.000 }
gfCNCPoint5[22091] = {X 450.4384, Y 41.0287, Z -7.1667, A 0.000, B 0.000, C 0.000 }
gfCNCPoint5[22092] = {X 450.4384, Y 34.2338, Z -7.1667, A 0.000, B 0.000, C 0.000 }
gfCNCPoint5[22093] = {X 447.3289, Y 34.2338, Z -7.1667, A 0.000, B 0.000, C 0.000 }
gfCNCPoint5[22094] = {X 442.9290, Y 42.8009, Z -7.1667, A 0.000, B 0.000, C 0.000 }
gfCNCPoint5[22095] = {X 442.9682, Y 42.9100, Z -7.1667, A 0.000, B 0.000, C 0.000 }
gfCNCPoint5[22096] = {X 443.1241, Y 43.5329, Z -7.1667, A 0.000, B 0.000, C 0.000 }
gfCNCPoint5[22097] = {X 443.1803, Y 44.1725, Z -7.1667, A 0.000, B 0.000, C 0.000 }
gfCNCPoint5[22098] = {X 443.1805, Y 45.0000, Z -7.1667, A 0.000, B 0.000, C 0.000 }
gfCNCPoint5[22099] = {X 443.0782, Y 45.9079, Z -7.1667, A 0.000, B 0.000, C 0.000 }
gfCNCPoint5[22100] = {X 442.7764, Y 46.7702, Z -7.1667, A 0.000, B 0.000, C 0.000 }
gfCNCPoint5[22101] = {X 442.2903, Y 47.5438, Z -7.1667, A 0.000, B 0.000, C 0.000 }
gfCNCPoint5[22102] = {X 441.6443, Y 48.1899, Z -7.1667, A 0.000, B 0.000, C 0.000 }
gfCNCPoint5[22103] = {X 440.8707, Y 48.6760, Z -7.1667, A 0.000, B 0.000, C 0.000 }
gfCNCPoint5[22104] = {X 440.0084, Y 48.9777, Z -7.1667, A 0.000, B 0.000, C 0.000 }
gfCNCPoint5[22105] = {X 439.1005, Y 49.0800, Z -7.1667, A 0.000, B 0.000, C 0.000 }
gfCNCPoint5[22106] = {X 432.5144, Y 49.0800, Z -7.1667, A 0.000, B 0.000, C 0.000 }
gfCNCPoint5[22107] = {X 431.6065, Y 48.9777, Z -7.1667, A 0.000, B 0.000, C 0.000 }
gfCNCPoint5[22108] = {X 430.7442, Y 48.6760, Z -7.1667, A 0.000, B 0.000, C 0.000 }
gfCNCPoint5[22109] = {X 429.9706, Y 48.1899, Z -7.1667, A 0.000, B 0.000, C 0.000 }
gfCNCPoint5[22110] = {X 429.3245, Y 47.5438, Z -7.1667, A 0.000, B 0.000, C 0.000 }
gfCNCPoint5[22111] = {X 428.8385, Y 46.7702, Z -7.1667, A 0.000, B 0.000, C 0.000 }
gfCNCPoint5[22112] = {X 428.5367, Y 45.9079, Z -7.1667, A 0.000, B 0.000, C 0.000 }
gfCNCPoint5[22113] = {X 428.4344, Y 45.0000, Z -7.1667, A 0.000, B 0.000, C 0.000 }
gfCNCPoint5[22114] = {X 428.4348, Y 44.1527, Z -7.1667, A 0.000, B 0.000, C 0.000 }
gfCNCPoint5[22115] = {X 428.5303, Y 43.3294, Z -7.1667, A 0.000, B 0.000, C 0.000 }
gfCNCPoint5[22116] = {X 428.7902, Y 42.5424, Z -7.1667, A 0.000, B 0.000, C 0.000 }
gfCNCPoint5[22117] = {X 429.2038, Y 41.8242, Z -7.1667, A 0.000, B 0.000, C 0.000 }
gfCNCPoint5[22118] = {X 429.7540, Y 41.2044, Z -7.1667, A 0.000, B 0.000, C 0.000 }
gfCNCPoint5[22119] = {X 430.4181, Y 40.7085, Z -7.1667, A 0.000, B 0.000, C 0.000 }
gfCNCPoint5[22120] = {X 431.1687, Y 40.3571, Z -7.1667, A 0.000, B 0.000, C 0.000 }
gfCNCPoint5[22121] = {X 435.3046, Y 32.2616, Z -7.1667, A 0.000, B 0.000, C 0.000 }
gfCNCPoint5[22122] = {X 434.1193, Y 31.4976, Z -7.1667, A 0.000, B 0.000, C 0.000 }
gfCNCPoint5[22123] = {X 433.0407, Y 30.5893, Z -7.1667, A 0.000, B 0.000, C 0.000 }
gfCNCPoint5[22124] = {X 432.0862, Y 29.5514, Z -7.1667, A 0.000, B 0.000, C 0.000 }
gfCNCPoint5[22125] = {X 431.2713, Y 28.4006, Z -7.1667, A 0.000, B 0.000, C 0.000 }
gfCNCPoint5[22126] = {X 430.6091, Y 27.1556, Z -7.1667, A 0.000, B 0.000, C 0.000 }
gfCNCPoint5[22127] = {X 430.1105, Y 25.8365, Z -7.1667, A 0.000, B 0.000, C 0.000 }
gfCNCPoint5[22128] = {X 429.6858, Y 24.0174, Z -7.1667, A 0.000, B 0.000, C 0.000 }
gfCNCPoint5[22129] = {X 429.4720, Y 22.1617, Z -7.1667, A 0.000, B 0.000, C 0.000 }
gfCNCPoint5[22130] = {X 429.4720, Y 20.2937, Z -7.1667, A 0.000, B 0.000, C 0.000 }
gfCNCPoint5[22131] = {X 429.6857, Y 18.4379, Z -7.1667, A 0.000, B 0.000, C 0.000 }
gfCNCPoint5[22132] = {X 430.1103, Y 16.6188, Z -7.1667, A 0.000, B 0.000, C 0.000 }
gfCNCPoint5[22133] = {X 430.6685, Y 15.1186, Z -7.1667, A 0.000, B 0.000, C 0.000 }
gfCNCPoint5[22134] = {X 431.4281, Y 13.7096, Z -7.1667, A 0.000, B 0.000, C 0.000 }
gfCNCPoint5[22135] = {X 432.3747, Y 12.4187, Z -7.1667, A 0.000, B 0.000, C 0.000 }
gfCNCPoint5[22136] = {X 433.4900, Y 11.2706, Z -7.1667, A 0.000, B 0.000, C 0.000 }
gfCNCPoint5[22137] = {X 434.7529, Y 10.2871, Z -7.1667, A 0.000, B 0.000, C 0.000 }
gfCNCPoint5[22138] = {X 436.1393, Y 9.4870, Z -7.1667, A 0.000, B 0.000, C 0.000 }
gfCNCPoint5[22139] = {X 437.6227, Y 8.8855, Z -7.1667, A 0.000, B 0.000, C 0.000 }
gfCNCPoint5[22140] = {X 439.1749, Y 8.4942, Z -7.1667, A 0.000, B 0.000, C 0.000 }
gfCNCPoint5[22141] = {X 441.2506, Y 8.2068, Z -7.1667, A 0.000, B 0.000, C 0.000 }
gfCNCPoint5[22142] = {X 443.3440, Y 8.1136, Z -7.1667, A 0.000, B 0.000, C 0.000 }
gfCNCPoint5[22143] = {X 444.0364, Y 8.1096, Z -7.1667, A 0.000, B 0.000, C 0.000 }
gfCNCPoint5[22144] = {X 459.4469, Y 8.1096, Z -7.1667, A 0.000, B 0.000, C 0.000 }
gfCNCPoint5[22145] = {X 460.3528, Y 8.2116, Z -7.1667, A 0.000, B 0.000, C 0.000 }
gfCNCPoint5[22146] = {X 461.2132, Y 8.5127, Z -7.1667, A 0.000, B 0.000, C 0.000 }
gfCNCPoint5[22147] = {X 461.9851, Y 8.9977, Z -7.1667, A 0.000, B 0.000, C 0.000 }
gfCNCPoint5[22148] = {X 462.6298, Y 9.6424, Z -7.1667, A 0.000, B 0.000, C 0.000 }
gfCNCPoint5[22149] = {X 463.1148, Y 10.4143, Z -7.1667, A 0.000, B 0.000, C 0.000 }
gfCNCPoint5[22150] = {X 463.4159, Y 11.2747, Z -7.1667, A 0.000, B 0.000, C 0.000 }
gfCNCPoint5[22151] = {X 463.5179, Y 12.1806, Z -7.1667, A 0.000, B 0.000, C 0.000 }
gfCNCPoint5[22152] = {X 463.5179, Y 12.9782, Z -7.1667, A 0.000, B 0.000, C 0.000 }
gfCNCPoint5[22153] = {X 463.4242, Y 13.8478, Z -7.1667, A 0.000, B 0.000, C 0.000 }
gfCNCPoint5[22154] = {X 463.1472, Y 14.6774, Z -7.1667, A 0.000, B 0.000, C 0.000 }
gfCNCPoint5[22155] = {X 462.6998, Y 15.4289, Z -7.1667, A 0.000, B 0.000, C 0.000 }
gfCNCPoint5[22156] = {X 462.1024, Y 16.0678, Z -7.1667, A 0.000, B 0.000, C 0.000 }
gfCNCPoint5[22157] = {X 462.0448, Y 16.1166, Z -7.1667, A 0.000, B 0.000, C 0.000 }
gfCNCPoint5[22158] = {X 461.9863, Y 16.1643, Z -7.1667, A 0.000, B 0.000, C 0.000 }
gfCNCPoint5[22159] = {X 461.9915, Y 16.1982, Z -7.1667, A 0.000, B 0.000, C 0.000 }
gfCNCPoint5[22160] = {X 461.9917, Y 28.5935, Z -7.1667, A 0.000, B 0.000, C 0.000 }
gfCNCPoint5[22161] = {X 465.9917, Y 28.5934, Z -7.1667, A 0.000, B 0.000, C 0.000 }
gfCNCPoint5[22162] = {X 465.9917, Y 28.5933, Z -7.1667, A 0.000, B 0.000, C 0.000 }
gfCNCPoint5[22163] = {X 461.9115, Y 28.5935, Z -7.1667, A 0.000, B 0.000, C 0.000 }
gfCNCPoint5[22164] = {X 461.9120, Y 41.0649, Z -7.1667, A 0.000, B 0.000, C 0.000 }
gfCNCPoint5[22165] = {X 462.0507, Y 41.1800, Z -7.1667, A 0.000, B 0.000, C 0.000 }
gfCNCPoint5[22166] = {X 462.6361, Y 41.8064, Z -7.1667, A 0.000, B 0.000, C 0.000 }
gfCNCPoint5[22167] = {X 463.0746, Y 42.5431, Z -7.1667, A 0.000, B 0.000, C 0.000 }
gfCNCPoint5[22168] = {X 463.3461, Y 43.3564, Z -7.1667, A 0.000, B 0.000, C 0.000 }
gfCNCPoint5[22169] = {X 463.4379, Y 44.2088, Z -7.1667, A 0.000, B 0.000, C 0.000 }
gfCNCPoint5[22170] = {X 463.4379, Y 45.0000, Z -7.1667, A 0.000, B 0.000, C 0.000 }
gfCNCPoint5[22171] = {X 463.3377, Y 45.8901, Z -7.1667, A 0.000, B 0.000, C 0.000 }
gfCNCPoint5[22172] = {X 463.0418, Y 46.7355, Z -7.1667, A 0.000, B 0.000, C 0.000 }
gfCNCPoint5[22173] = {X 462.5653, Y 47.4940, Z -7.1667, A 0.000, B 0.000, C 0.000 }
gfCNCPoint5[22174] = {X 461.9319, Y 48.1273, Z -7.1667, A 0.000, B 0.000, C 0.000 }
gfCNCPoint5[22175] = {X 461.1735, Y 48.6039, Z -7.1667, A 0.000, B 0.000, C 0.000 }
gfCNCPoint5[22176] = {X 460.3280, Y 48.8997, Z -7.1667, A 0.000, B 0.000, C 0.000 }
gfCNCPoint5[22177] = {X 459.4379, Y 49.0000, Z -7.1667, A 0.000, B 0.000, C 0.000 }
gfCNCPoint5[22178] = {X 452.9945, Y 49.0000, Z -7.1667, A 0.000, B 0.000, C 0.000 }
gfCNCPoint5[22179] = {X 452.1044, Y 48.8997, Z -7.1667, A 0.000, B 0.000, C 0.000 }
gfCNCPoint5[22180] = {X 451.2589, Y 48.6039, Z -7.1667, A 0.000, B 0.000, C 0.000 }
gfCNCPoint5[22181] = {X 450.5005, Y 48.1273, Z -7.1667, A 0.000, B 0.000, C 0.000 }
gfCNCPoint5[22182] = {X 449.8671, Y 47.4939, Z -7.1667, A 0.000, B 0.000, C 0.000 }
gfCNCPoint5[22183] = {X 449.3906, Y 46.7355, Z -7.1667, A 0.000, B 0.000, C 0.000 }
gfCNCPoint5[22184] = {X 449.0948, Y 45.8901, Z -7.1667, A 0.000, B 0.000, C 0.000 }
gfCNCPoint5[22185] = {X 448.9945, Y 45.0000, Z -7.1667, A 0.000, B 0.000, C 0.000 }
gfCNCPoint5[22186] = {X 448.9949, Y 44.1538, Z -7.1667, A 0.000, B 0.000, C 0.000 }
gfCNCPoint5[22187] = {X 449.1055, Y 43.2730, Z -7.1667, A 0.000, B 0.000, C 0.000 }
gfCNCPoint5[22188] = {X 449.4077, Y 42.4382, Z -7.1667, A 0.000, B 0.000, C 0.000 }
gfCNCPoint5[22189] = {X 449.8865, Y 41.6907, Z -7.1667, A 0.000, B 0.000, C 0.000 }
gfCNCPoint5[22190] = {X 450.5184, Y 41.0672, Z -7.1667, A 0.000, B 0.000, C 0.000 }
gfCNCPoint5[22191] = {X 450.5184, Y 34.1538, Z -7.1667, A 0.000, B 0.000, C 0.000 }
gfCNCPoint5[22192] = {X 447.2801, Y 34.1538, Z -7.1667, A 0.000, B 0.000, C 0.000 }
gfCNCPoint5[22193] = {X 442.8420, Y 42.7952, Z -7.1667, A 0.000, B 0.000, C 0.000 }
gfCNCPoint5[22194] = {X 442.8972, Y 42.9499, Z -7.1667, A 0.000, B 0.000, C 0.000 }
gfCNCPoint5[22195] = {X 443.0493, Y 43.5712, Z -7.1667, A 0.000, B 0.000, C 0.000 }
gfCNCPoint5[22196] = {X 443.1005, Y 44.2089, Z -7.1667, A 0.000, B 0.000, C 0.000 }
gfCNCPoint5[22197] = {X 443.1005, Y 45.0000, Z -7.1667, A 0.000, B 0.000, C 0.000 }
gfCNCPoint5[22198] = {X 443.0002, Y 45.8901, Z -7.1667, A 0.000, B 0.000, C 0.000 }
gfCNCPoint5[22199] = {X 442.7043, Y 46.7355, Z -7.1667, A 0.000, B 0.000, C 0.000 }
gfCNCPoint5[22200] = {X 442.2278, Y 47.4940, Z -7.1667, A 0.000, B 0.000, C 0.000 }
gfCNCPoint5[22201] = {X 441.5944, Y 48.1273, Z -7.1667, A 0.000, B 0.000, C 0.000 }
gfCNCPoint5[22202] = {X 440.8360, Y 48.6039, Z -7.1667, A 0.000, B 0.000, C 0.000 }
gfCNCPoint5[22203] = {X 439.9906, Y 48.8997, Z -7.1667, A 0.000, B 0.000, C 0.000 }
gfCNCPoint5[22204] = {X 439.1005, Y 49.0000, Z -7.1667, A 0.000, B 0.000, C 0.000 }
gfCNCPoint5[22205] = {X 432.5144, Y 49.0000, Z -7.1667, A 0.000, B 0.000, C 0.000 }
gfCNCPoint5[22206] = {X 431.6243, Y 48.8997, Z -7.1667, A 0.000, B 0.000, C 0.000 }
gfCNCPoint5[22207] = {X 430.7789, Y 48.6039, Z -7.1667, A 0.000, B 0.000, C 0.000 }
gfCNCPoint5[22208] = {X 430.0204, Y 48.1273, Z -7.1667, A 0.000, B 0.000, C 0.000 }
gfCNCPoint5[22209] = {X 429.3871, Y 47.4940, Z -7.1667, A 0.000, B 0.000, C 0.000 }
gfCNCPoint5[22210] = {X 428.9105, Y 46.7355, Z -7.1667, A 0.000, B 0.000, C 0.000 }
gfCNCPoint5[22211] = {X 428.6147, Y 45.8901, Z -7.1667, A 0.000, B 0.000, C 0.000 }
gfCNCPoint5[22212] = {X 428.5144, Y 45.0000, Z -7.1667, A 0.000, B 0.000, C 0.000 }
gfCNCPoint5[22213] = {X 428.5148, Y 44.1538, Z -7.1667, A 0.000, B 0.000, C 0.000 }
gfCNCPoint5[22214] = {X 428.6096, Y 43.3414, Z -7.1667, A 0.000, B 0.000, C 0.000 }
gfCNCPoint5[22215] = {X 428.8676, Y 42.5654, Z -7.1667, A 0.000, B 0.000, C 0.000 }
gfCNCPoint5[22216] = {X 429.2781, Y 41.8580, Z -7.1667, A 0.000, B 0.000, C 0.000 }
gfCNCPoint5[22217] = {X 429.8239, Y 41.2489, Z -7.1667, A 0.000, B 0.000, C 0.000 }
gfCNCPoint5[22218] = {X 430.4821, Y 40.7635, Z -7.1667, A 0.000, B 0.000, C 0.000 }
gfCNCPoint5[22219] = {X 431.2253, Y 40.4222, Z -7.1667, A 0.000, B 0.000, C 0.000 }
gfCNCPoint5[22220] = {X 435.4111, Y 32.2290, Z -7.1667, A 0.000, B 0.000, C 0.000 }
gfCNCPoint5[22221] = {X 434.2187, Y 31.4713, Z -7.1667, A 0.000, B 0.000, C 0.000 }
gfCNCPoint5[22222] = {X 433.1333, Y 30.5670, Z -7.1667, A 0.000, B 0.000, C 0.000 }
gfCNCPoint5[22223] = {X 432.1727, Y 29.5310, Z -7.1667, A 0.000, B 0.000, C 0.000 }
gfCNCPoint5[22224] = {X 431.3529, Y 28.3804, Z -7.1667, A 0.000, B 0.000, C 0.000 }
gfCNCPoint5[22225] = {X 430.6873, Y 27.1343, Z -7.1667, A 0.000, B 0.000, C 0.000 }
gfCNCPoint5[22226] = {X 430.1870, Y 25.8131, Z -7.1667, A 0.000, B 0.000, C 0.000 }
gfCNCPoint5[22227] = {X 429.7645, Y 24.0030, Z -7.1667, A 0.000, B 0.000, C 0.000 }
gfCNCPoint5[22228] = {X 429.5519, Y 22.1566, Z -7.1667, A 0.000, B 0.000, C 0.000 }
gfCNCPoint5[22229] = {X 429.5519, Y 20.2979, Z -7.1667, A 0.000, B 0.000, C 0.000 }
gfCNCPoint5[22230] = {X 429.7645, Y 18.4514, Z -7.1667, A 0.000, B 0.000, C 0.000 }
gfCNCPoint5[22231] = {X 430.1870, Y 16.6414, Z -7.1667, A 0.000, B 0.000, C 0.000 }
gfCNCPoint5[22232] = {X 430.7414, Y 15.1515, Z -7.1667, A 0.000, B 0.000, C 0.000 }
gfCNCPoint5[22233] = {X 431.4958, Y 13.7523, Z -7.1667, A 0.000, B 0.000, C 0.000 }
gfCNCPoint5[22234] = {X 432.4358, Y 12.4703, Z -7.1667, A 0.000, B 0.000, C 0.000 }
gfCNCPoint5[22235] = {X 433.5435, Y 11.3301, Z -7.1667, A 0.000, B 0.000, C 0.000 }
gfCNCPoint5[22236] = {X 434.7978, Y 10.3534, Z -7.1667, A 0.000, B 0.000, C 0.000 }
gfCNCPoint5[22237] = {X 436.1746, Y 9.5588, Z -7.1667, A 0.000, B 0.000, C 0.000 }
gfCNCPoint5[22238] = {X 437.6478, Y 8.9615, Z -7.1667, A 0.000, B 0.000, C 0.000 }
gfCNCPoint5[22239] = {X 439.1893, Y 8.5729, Z -7.1667, A 0.000, B 0.000, C 0.000 }
gfCNCPoint5[22240] = {X 441.2579, Y 8.2864, Z -7.1667, A 0.000, B 0.000, C 0.000 }
gfCNCPoint5[22241] = {X 443.3442, Y 8.1936, Z -7.1667, A 0.000, B 0.000, C 0.000 }
gfCNCPoint5[22242] = {X 444.0367, Y 8.1896, Z -7.1667, A 0.000, B 0.000, C 0.000 }
gfCNCPoint5[22243] = {X 459.4469, Y 8.1896, Z -7.1667, A 0.000, B 0.000, C 0.000 }
gfCNCPoint5[22244] = {X 460.3350, Y 8.2896, Z -7.1667, A 0.000, B 0.000, C 0.000 }
gfCNCPoint5[22245] = {X 461.1785, Y 8.5848, Z -7.1667, A 0.000, B 0.000, C 0.000 }
gfCNCPoint5[22246] = {X 461.9353, Y 9.0603, Z -7.1667, A 0.000, B 0.000, C 0.000 }
gfCNCPoint5[22247] = {X 462.5672, Y 9.6922, Z -7.1667, A 0.000, B 0.000, C 0.000 }
gfCNCPoint5[22248] = {X 463.0427, Y 10.4490, Z -7.1667, A 0.000, B 0.000, C 0.000 }
gfCNCPoint5[22249] = {X 463.3379, Y 11.2925, Z -7.1667, A 0.000, B 0.000, C 0.000 }
gfCNCPoint5[22250] = {X 463.4379, Y 12.1806, Z -7.1667, A 0.000, B 0.000, C 0.000 }
gfCNCPoint5[22251] = {X 463.4378, Y 13.0163, Z -7.1667, A 0.000, B 0.000, C 0.000 }
gfCNCPoint5[22252] = {X 463.3398, Y 13.8586, Z -7.1667, A 0.000, B 0.000, C 0.000 }
gfCNCPoint5[22253] = {X 463.0665, Y 14.6614, Z -7.1667, A 0.000, B 0.000, C 0.000 }
gfCNCPoint5[22254] = {X 462.6301, Y 15.3885, Z -7.1667, A 0.000, B 0.000, C 0.000 }
gfCNCPoint5[22255] = {X 462.0502, Y 16.0072, Z -7.1667, A 0.000, B 0.000, C 0.000 }
gfCNCPoint5[22256] = {X 461.9730, Y 16.0721, Z -7.1667, A 0.000, B 0.000, C 0.000 }
gfCNCPoint5[22257] = {X 461.8942, Y 16.1351, Z -7.1667, A 0.000, B 0.000, C 0.000 }
gfCNCPoint5[22258] = {X 461.9115, Y 16.1934, Z -7.1667, A 0.000, B 0.000, C 0.000 }
gfCNCPoint5[22259] = {X 461.9110, Y 16.7687, Z -7.1667, A 0.000, B 0.000, C 0.000 }
gfCNCPoint5[22260] = {X 461.9115, Y 28.5935, Z -7.1667, A 0.000, B 0.000, C 0.000 }
gfCNCPoint5[22261] = {X 465.9917, Y 28.5933, Z -7.1667, A 0.000, B 0.000, C 0.000 }
gfCNCPoint5[22262] = {X 465.9917, Y 28.5933, Z -4.1667, A 0.000, B 0.000, C 0.000 }
gfCNCPoint5[22263] = {X 465.9917, Y 28.5933, Z 11.0000, A 0.000, B 0.000, C 0.000 }
gfCNCPoint5[22264] = {X 492.3835, Y 3.7896, Z 11.0000, A 0.000, B 0.000, C 0.000 }
gfCNCPoint5[22265] = {X 492.3835, Y 3.7896, Z -4.1667, A 0.000, B 0.000, C 0.000 }
gfCNCPoint5[22266] = {X 492.3835, Y 3.7896, Z -7.1667, A 0.000, B 0.000, C 0.000 }
gfCNCPoint5[22267] = {X 492.3835, Y 7.8696, Z -7.1667, A 0.000, B 0.000, C 0.000 }
gfCNCPoint5[22268] = {X 502.2066, Y 7.8696, Z -7.1667, A 0.000, B 0.000, C 0.000 }
gfCNCPoint5[22269] = {X 502.7395, Y 7.8737, Z -7.1667, A 0.000, B 0.000, C 0.000 }
gfCNCPoint5[22270] = {X 503.6913, Y 7.9880, Z -7.1667, A 0.000, B 0.000, C 0.000 }
gfCNCPoint5[22271] = {X 504.5943, Y 8.3102, Z -7.1667, A 0.000, B 0.000, C 0.000 }
gfCNCPoint5[22272] = {X 505.4035, Y 8.8243, Z -7.1667, A 0.000, B 0.000, C 0.000 }
gfCNCPoint5[22273] = {X 506.0788, Y 9.5049, Z -7.1667, A 0.000, B 0.000, C 0.000 }
gfCNCPoint5[22274] = {X 506.5866, Y 10.3180, Z -7.1667, A 0.000, B 0.000, C 0.000 }
gfCNCPoint5[22275] = {X 506.9017, Y 11.2235, Z -7.1667, A 0.000, B 0.000, C 0.000 }
gfCNCPoint5[22276] = {X 507.0085, Y 12.1762, Z -7.1667, A 0.000, B 0.000, C 0.000 }
gfCNCPoint5[22277] = {X 507.0085, Y 12.9782, Z -7.1667, A 0.000, B 0.000, C 0.000 }
gfCNCPoint5[22278] = {X 506.9072, Y 13.9079, Z -7.1667, A 0.000, B 0.000, C 0.000 }
gfCNCPoint5[22279] = {X 506.6082, Y 14.7940, Z -7.1667, A 0.000, B 0.000, C 0.000 }
gfCNCPoint5[22280] = {X 506.1256, Y 15.5951, Z -7.1667, A 0.000, B 0.000, C 0.000 }
gfCNCPoint5[22281] = {X 505.4818, Y 16.2734, Z -7.1667, A 0.000, B 0.000, C 0.000 }
gfCNCPoint5[22282] = {X 505.4821, Y 40.9136, Z -7.1667, A 0.000, B 0.000, C 0.000 }
gfCNCPoint5[22283] = {X 506.1201, Y 41.5845, Z -7.1667, A 0.000, B 0.000, C 0.000 }
gfCNCPoint5[22284] = {X 506.6004, Y 42.3760, Z -7.1667, A 0.000, B 0.000, C 0.000 }
gfCNCPoint5[22285] = {X 506.9011, Y 43.2517, Z -7.1667, A 0.000, B 0.000, C 0.000 }
gfCNCPoint5[22286] = {X 507.0083, Y 44.1713, Z -7.1667, A 0.000, B 0.000, C 0.000 }
gfCNCPoint5[22287] = {X 507.0085, Y 45.0000, Z -7.1667, A 0.000, B 0.000, C 0.000 }
gfCNCPoint5[22288] = {X 506.9002, Y 45.9613, Z -7.1667, A 0.000, B 0.000, C 0.000 }
gfCNCPoint5[22289] = {X 506.5807, Y 46.8744, Z -7.1667, A 0.000, B 0.000, C 0.000 }
gfCNCPoint5[22290] = {X 506.0660, Y 47.6935, Z -7.1667, A 0.000, B 0.000, C 0.000 }
gfCNCPoint5[22291] = {X 505.3820, Y 48.3775, Z -7.1667, A 0.000, B 0.000, C 0.000 }
gfCNCPoint5[22292] = {X 504.5629, Y 48.8922, Z -7.1667, A 0.000, B 0.000, C 0.000 }
gfCNCPoint5[22293] = {X 503.6498, Y 49.2117, Z -7.1667, A 0.000, B 0.000, C 0.000 }
gfCNCPoint5[22294] = {X 502.6885, Y 49.3200, Z -7.1667, A 0.000, B 0.000, C 0.000 }
gfCNCPoint5[22295] = {X 496.2450, Y 49.3200, Z -7.1667, A 0.000, B 0.000, C 0.000 }
gfCNCPoint5[22296] = {X 495.2885, Y 49.2128, Z -7.1667, A 0.000, B 0.000, C 0.000 }
gfCNCPoint5[22297] = {X 494.3794, Y 48.8964, Z -7.1667, A 0.000, B 0.000, C 0.000 }
gfCNCPoint5[22298] = {X 493.5630, Y 48.3866, Z -7.1667, A 0.000, B 0.000, C 0.000 }
gfCNCPoint5[22299] = {X 492.8797, Y 47.7087, Z -7.1667, A 0.000, B 0.000, C 0.000 }
gfCNCPoint5[22300] = {X 492.3635, Y 46.8963, Z -7.1667, A 0.000, B 0.000, C 0.000 }
gfCNCPoint5[22301] = {X 492.0399, Y 45.9898, Z -7.1667, A 0.000, B 0.000, C 0.000 }
gfCNCPoint5[22302] = {X 491.9252, Y 45.0341, Z -7.1667, A 0.000, B 0.000, C 0.000 }
gfCNCPoint5[22303] = {X 491.9254, Y 44.1494, Z -7.1667, A 0.000, B 0.000, C 0.000 }
gfCNCPoint5[22304] = {X 492.0359, Y 43.2364, Z -7.1667, A 0.000, B 0.000, C 0.000 }
gfCNCPoint5[22305] = {X 492.3371, Y 42.3675, Z -7.1667, A 0.000, B 0.000, C 0.000 }
gfCNCPoint5[22306] = {X 492.8153, Y 41.5821, Z -7.1667, A 0.000, B 0.000, C 0.000 }
gfCNCPoint5[22307] = {X 493.4490, Y 40.9157, Z -7.1667, A 0.000, B 0.000, C 0.000 }
gfCNCPoint5[22308] = {X 493.4490, Y 34.4738, Z -7.1667, A 0.000, B 0.000, C 0.000 }
gfCNCPoint5[22309] = {X 490.7254, Y 34.4738, Z -7.1667, A 0.000, B 0.000, C 0.000 }
gfCNCPoint5[22310] = {X 486.4406, Y 42.8179, Z -7.1667, A 0.000, B 0.000, C 0.000 }
gfCNCPoint5[22311] = {X 486.4454, Y 42.8308, Z -7.1667, A 0.000, B 0.000, C 0.000 }
gfCNCPoint5[22312] = {X 486.6110, Y 43.4914, Z -7.1667, A 0.000, B 0.000, C 0.000 }
gfCNCPoint5[22313] = {X 486.6708, Y 44.1699, Z -7.1667, A 0.000, B 0.000, C 0.000 }
gfCNCPoint5[22314] = {X 486.6710, Y 45.0000, Z -7.1667, A 0.000, B 0.000, C 0.000 }
gfCNCPoint5[22315] = {X 486.5627, Y 45.9613, Z -7.1667, A 0.000, B 0.000, C 0.000 }
gfCNCPoint5[22316] = {X 486.2432, Y 46.8744, Z -7.1667, A 0.000, B 0.000, C 0.000 }
gfCNCPoint5[22317] = {X 485.7285, Y 47.6935, Z -7.1667, A 0.000, B 0.000, C 0.000 }
gfCNCPoint5[22318] = {X 485.0445, Y 48.3775, Z -7.1667, A 0.000, B 0.000, C 0.000 }
gfCNCPoint5[22319] = {X 484.2254, Y 48.8922, Z -7.1667, A 0.000, B 0.000, C 0.000 }
gfCNCPoint5[22320] = {X 483.3123, Y 49.2117, Z -7.1667, A 0.000, B 0.000, C 0.000 }
gfCNCPoint5[22321] = {X 482.3510, Y 49.3200, Z -7.1667, A 0.000, B 0.000, C 0.000 }
gfCNCPoint5[22322] = {X 475.7650, Y 49.3200, Z -7.1667, A 0.000, B 0.000, C 0.000 }
gfCNCPoint5[22323] = {X 474.8037, Y 49.2117, Z -7.1667, A 0.000, B 0.000, C 0.000 }
gfCNCPoint5[22324] = {X 473.8906, Y 48.8922, Z -7.1667, A 0.000, B 0.000, C 0.000 }
gfCNCPoint5[22325] = {X 473.0715, Y 48.3775, Z -7.1667, A 0.000, B 0.000, C 0.000 }
gfCNCPoint5[22326] = {X 472.3875, Y 47.6935, Z -7.1667, A 0.000, B 0.000, C 0.000 }
gfCNCPoint5[22327] = {X 471.8728, Y 46.8745, Z -7.1667, A 0.000, B 0.000, C 0.000 }
gfCNCPoint5[22328] = {X 471.5533, Y 45.9614, Z -7.1667, A 0.000, B 0.000, C 0.000 }
gfCNCPoint5[22329] = {X 471.4450, Y 45.0001, Z -7.1667, A 0.000, B 0.000, C 0.000 }
gfCNCPoint5[22330] = {X 471.4454, Y 44.1494, Z -7.1667, A 0.000, B 0.000, C 0.000 }
gfCNCPoint5[22331] = {X 471.5430, Y 43.2935, Z -7.1667, A 0.000, B 0.000, C 0.000 }
gfCNCPoint5[22332] = {X 471.8086, Y 42.4740, Z -7.1667, A 0.000, B 0.000, C 0.000 }
gfCNCPoint5[22333] = {X 472.2314, Y 41.7236, Z -7.1667, A 0.000, B 0.000, C 0.000 }
gfCNCPoint5[22334] = {X 472.7947, Y 41.0719, Z -7.1667, A 0.000, B 0.000, C 0.000 }
gfCNCPoint5[22335] = {X 473.4762, Y 40.5449, Z -7.1667, A 0.000, B 0.000, C 0.000 }
gfCNCPoint5[22336] = {X 474.2486, Y 40.1637, Z -7.1667, A 0.000, B 0.000, C 0.000 }
gfCNCPoint5[22337] = {X 478.2330, Y 32.3647, Z -7.1667, A 0.000, B 0.000, C 0.000 }
gfCNCPoint5[22338] = {X 476.9688, Y 31.4977, Z -7.1667, A 0.000, B 0.000, C 0.000 }
gfCNCPoint5[22339] = {X 475.8317, Y 30.4696, Z -7.1667, A 0.000, B 0.000, C 0.000 }
gfCNCPoint5[22340] = {X 474.8421, Y 29.2989, Z -7.1667, A 0.000, B 0.000, C 0.000 }
gfCNCPoint5[22341] = {X 474.0178, Y 28.0065, Z -7.1667, A 0.000, B 0.000, C 0.000 }
gfCNCPoint5[22342] = {X 473.3733, Y 26.6156, Z -7.1667, A 0.000, B 0.000, C 0.000 }
gfCNCPoint5[22343] = {X 472.9204, Y 25.1511, Z -7.1667, A 0.000, B 0.000, C 0.000 }
gfCNCPoint5[22344] = {X 472.6067, Y 23.4679, Z -7.1667, A 0.000, B 0.000, C 0.000 }
gfCNCPoint5[22345] = {X 472.4665, Y 21.7616, Z -7.1667, A 0.000, B 0.000, C 0.000 }
gfCNCPoint5[22346] = {X 472.5012, Y 20.0498, Z -7.1667, A 0.000, B 0.000, C 0.000 }
gfCNCPoint5[22347] = {X 472.7104, Y 18.3506, Z -7.1667, A 0.000, B 0.000, C 0.000 }
gfCNCPoint5[22348] = {X 473.0921, Y 16.6815, Z -7.1667, A 0.000, B 0.000, C 0.000 }
gfCNCPoint5[22349] = {X 473.6351, Y 15.1666, Z -7.1667, A 0.000, B 0.000, C 0.000 }
gfCNCPoint5[22350] = {X 474.3786, Y 13.7393, Z -7.1667, A 0.000, B 0.000, C 0.000 }
gfCNCPoint5[22351] = {X 475.3088, Y 12.4261, Z -7.1667, A 0.000, B 0.000, C 0.000 }
gfCNCPoint5[22352] = {X 476.4086, Y 11.2512, Z -7.1667, A 0.000, B 0.000, C 0.000 }
gfCNCPoint5[22353] = {X 477.6576, Y 10.2364, Z -7.1667, A 0.000, B 0.000, C 0.000 }
gfCNCPoint5[22354] = {X 479.0327, Y 9.4005, Z -7.1667, A 0.000, B 0.000, C 0.000 }
gfCNCPoint5[22355] = {X 480.5086, Y 8.7588, Z -7.1667, A 0.000, B 0.000, C 0.000 }
gfCNCPoint5[22356] = {X 482.0578, Y 8.3232, Z -7.1667, A 0.000, B 0.000, C 0.000 }
gfCNCPoint5[22357] = {X 484.1552, Y 7.9968, Z -7.1667, A 0.000, B 0.000, C 0.000 }
gfCNCPoint5[22358] = {X 486.2746, Y 7.8817, Z -7.1667, A 0.000, B 0.000, C 0.000 }
gfCNCPoint5[22359] = {X 486.9679, Y 7.8696, Z -7.1667, A 0.000, B 0.000, C 0.000 }
gfCNCPoint5[22360] = {X 492.3835, Y 7.8696, Z -7.1667, A 0.000, B 0.000, C 0.000 }
gfCNCPoint5[22361] = {X 492.3835, Y 3.8696, Z -7.1667, A 0.000, B 0.000, C 0.000 }
gfCNCPoint5[22362] = {X 492.3835, Y 7.9496, Z -7.1667, A 0.000, B 0.000, C 0.000 }
gfCNCPoint5[22363] = {X 502.2063, Y 7.9496, Z -7.1667, A 0.000, B 0.000, C 0.000 }
gfCNCPoint5[22364] = {X 502.7388, Y 7.9537, Z -7.1667, A 0.000, B 0.000, C 0.000 }
gfCNCPoint5[22365] = {X 503.6730, Y 8.0659, Z -7.1667, A 0.000, B 0.000, C 0.000 }
gfCNCPoint5[22366] = {X 504.5592, Y 8.3821, Z -7.1667, A 0.000, B 0.000, C 0.000 }
gfCNCPoint5[22367] = {X 505.3533, Y 8.8866, Z -7.1667, A 0.000, B 0.000, C 0.000 }
gfCNCPoint5[22368] = {X 506.0160, Y 9.5545, Z -7.1667, A 0.000, B 0.000, C 0.000 }
gfCNCPoint5[22369] = {X 506.5144, Y 10.3526, Z -7.1667, A 0.000, B 0.000, C 0.000 }
gfCNCPoint5[22370] = {X 506.8237, Y 11.2412, Z -7.1667, A 0.000, B 0.000, C 0.000 }
gfCNCPoint5[22371] = {X 506.9285, Y 12.1762, Z -7.1667, A 0.000, B 0.000, C 0.000 }
gfCNCPoint5[22372] = {X 506.9285, Y 12.9782, Z -7.1667, A 0.000, B 0.000, C 0.000 }
gfCNCPoint5[22373] = {X 506.8271, Y 13.8997, Z -7.1667, A 0.000, B 0.000, C 0.000 }
gfCNCPoint5[22374] = {X 506.5279, Y 14.7771, Z -7.1667, A 0.000, B 0.000, C 0.000 }
gfCNCPoint5[22375] = {X 506.0451, Y 15.5686, Z -7.1667, A 0.000, B 0.000, C 0.000 }
gfCNCPoint5[22376] = {X 505.4018, Y 16.2362, Z -7.1667, A 0.000, B 0.000, C 0.000 }
gfCNCPoint5[22377] = {X 505.4021, Y 40.9512, Z -7.1667, A 0.000, B 0.000, C 0.000 }
gfCNCPoint5[22378] = {X 505.4303, Y 40.9746, Z -7.1667, A 0.000, B 0.000, C 0.000 }
gfCNCPoint5[22379] = {X 506.0565, Y 41.6331, Z -7.1667, A 0.000, B 0.000, C 0.000 }
gfCNCPoint5[22380] = {X 506.5280, Y 42.4100, Z -7.1667, A 0.000, B 0.000, C 0.000 }
gfCNCPoint5[22381] = {X 506.8231, Y 43.2694, Z -7.1667, A 0.000, B 0.000, C 0.000 }
gfCNCPoint5[22382] = {X 506.9283, Y 44.1720, Z -7.1667, A 0.000, B 0.000, C 0.000 }
gfCNCPoint5[22383] = {X 506.9285, Y 45.0000, Z -7.1667, A 0.000, B 0.000, C 0.000 }
gfCNCPoint5[22384] = {X 506.8222, Y 45.9435, Z -7.1667, A 0.000, B 0.000, C 0.000 }
gfCNCPoint5[22385] = {X 506.5086, Y 46.8397, Z -7.1667, A 0.000, B 0.000, C 0.000 }
gfCNCPoint5[22386] = {X 506.0035, Y 47.6436, Z -7.1667, A 0.000, B 0.000, C 0.000 }
gfCNCPoint5[22387] = {X 505.3321, Y 48.3150, Z -7.1667, A 0.000, B 0.000, C 0.000 }
gfCNCPoint5[22388] = {X 504.5282, Y 48.8201, Z -7.1667, A 0.000, B 0.000, C 0.000 }
gfCNCPoint5[22389] = {X 503.6320, Y 49.1337, Z -7.1667, A 0.000, B 0.000, C 0.000 }
gfCNCPoint5[22390] = {X 502.6885, Y 49.2400, Z -7.1667, A 0.000, B 0.000, C 0.000 }
gfCNCPoint5[22391] = {X 496.2450, Y 49.2400, Z -7.1667, A 0.000, B 0.000, C 0.000 }
gfCNCPoint5[22392] = {X 495.3062, Y 49.1348, Z -7.1667, A 0.000, B 0.000, C 0.000 }
gfCNCPoint5[22393] = {X 494.4140, Y 48.8242, Z -7.1667, A 0.000, B 0.000, C 0.000 }
gfCNCPoint5[22394] = {X 493.6127, Y 48.3239, Z -7.1667, A 0.000, B 0.000, C 0.000 }
gfCNCPoint5[22395] = {X 492.9420, Y 47.6585, Z -7.1667, A 0.000, B 0.000, C 0.000 }
gfCNCPoint5[22396] = {X 492.4354, Y 46.8612, Z -7.1667, A 0.000, B 0.000, C 0.000 }
gfCNCPoint5[22397] = {X 492.1178, Y 45.9714, Z -7.1667, A 0.000, B 0.000, C 0.000 }
gfCNCPoint5[22398] = {X 492.0052, Y 45.0335, Z -7.1667, A 0.000, B 0.000, C 0.000 }
gfCNCPoint5[22399] = {X 492.0054, Y 44.1505, Z -7.1667, A 0.000, B 0.000, C 0.000 }
gfCNCPoint5[22400] = {X 492.1159, Y 43.2454, Z -7.1667, A 0.000, B 0.000, C 0.000 }
gfCNCPoint5[22401] = {X 492.4173, Y 42.3850, Z -7.1667, A 0.000, B 0.000, C 0.000 }
gfCNCPoint5[22402] = {X 492.8957, Y 41.6088, Z -7.1667, A 0.000, B 0.000, C 0.000 }
gfCNCPoint5[22403] = {X 493.5290, Y 40.9529, Z -7.1667, A 0.000, B 0.000, C 0.000 }
gfCNCPoint5[22404] = {X 493.5290, Y 34.3938, Z -7.1667, A 0.000, B 0.000, C 0.000 }
gfCNCPoint5[22405] = {X 490.6766, Y 34.3938, Z -7.1667, A 0.000, B 0.000, C 0.000 }
gfCNCPoint5[22406] = {X 486.3534, Y 42.8126, Z -7.1667, A 0.000, B 0.000, C 0.000 }
gfCNCPoint5[22407] = {X 486.3699, Y 42.8574, Z -7.1667, A 0.000, B 0.000, C 0.000 }
gfCNCPoint5[22408] = {X 486.5322, Y 43.5053, Z -7.1667, A 0.000, B 0.000, C 0.000 }
gfCNCPoint5[22409] = {X 486.5908, Y 44.1706, Z -7.1667, A 0.000, B 0.000, C 0.000 }
gfCNCPoint5[22410] = {X 486.5910, Y 45.0000, Z -7.1667, A 0.000, B 0.000, C 0.000 }
gfCNCPoint5[22411] = {X 486.4847, Y 45.9435, Z -7.1667, A 0.000, B 0.000, C 0.000 }
gfCNCPoint5[22412] = {X 486.1711, Y 46.8397, Z -7.1667, A 0.000, B 0.000, C 0.000 }
gfCNCPoint5[22413] = {X 485.6660, Y 47.6436, Z -7.1667, A 0.000, B 0.000, C 0.000 }
gfCNCPoint5[22414] = {X 484.9946, Y 48.3150, Z -7.1667, A 0.000, B 0.000, C 0.000 }
gfCNCPoint5[22415] = {X 484.1907, Y 48.8201, Z -7.1667, A 0.000, B 0.000, C 0.000 }
gfCNCPoint5[22416] = {X 483.2945, Y 49.1337, Z -7.1667, A 0.000, B 0.000, C 0.000 }
gfCNCPoint5[22417] = {X 482.3510, Y 49.2400, Z -7.1667, A 0.000, B 0.000, C 0.000 }
gfCNCPoint5[22418] = {X 475.7650, Y 49.2400, Z -7.1667, A 0.000, B 0.000, C 0.000 }
gfCNCPoint5[22419] = {X 474.8215, Y 49.1337, Z -7.1667, A 0.000, B 0.000, C 0.000 }
gfCNCPoint5[22420] = {X 473.9253, Y 48.8201, Z -7.1667, A 0.000, B 0.000, C 0.000 }
gfCNCPoint5[22421] = {X 473.1214, Y 48.3150, Z -7.1667, A 0.000, B 0.000, C 0.000 }
gfCNCPoint5[22422] = {X 472.4500, Y 47.6436, Z -7.1667, A 0.000, B 0.000, C 0.000 }
gfCNCPoint5[22423] = {X 471.9449, Y 46.8397, Z -7.1667, A 0.000, B 0.000, C 0.000 }
gfCNCPoint5[22424] = {X 471.6313, Y 45.9436, Z -7.1667, A 0.000, B 0.000, C 0.000 }
gfCNCPoint5[22425] = {X 471.5250, Y 45.0001, Z -7.1667, A 0.000, B 0.000, C 0.000 }
gfCNCPoint5[22426] = {X 471.5254, Y 44.1505, Z -7.1667, A 0.000, B 0.000, C 0.000 }
gfCNCPoint5[22427] = {X 471.6223, Y 43.3054, Z -7.1667, A 0.000, B 0.000, C 0.000 }
gfCNCPoint5[22428] = {X 471.8860, Y 42.4967, Z -7.1667, A 0.000, B 0.000, C 0.000 }
gfCNCPoint5[22429] = {X 472.3057, Y 41.7570, Z -7.1667, A 0.000, B 0.000, C 0.000 }
gfCNCPoint5[22430] = {X 472.8647, Y 41.1158, Z -7.1667, A 0.000, B 0.000, C 0.000 }
gfCNCPoint5[22431] = {X 473.5404, Y 40.5992, Z -7.1667, A 0.000, B 0.000, C 0.000 }
gfCNCPoint5[22432] = {X 474.3057, Y 40.2278, Z -7.1667, A 0.000, B 0.000, C 0.000 }
gfCNCPoint5[22433] = {X 478.3385, Y 32.3339, Z -7.1667, A 0.000, B 0.000, C 0.000 }
gfCNCPoint5[22434] = {X 477.0676, Y 31.4735, Z -7.1667, A 0.000, B 0.000, C 0.000 }
gfCNCPoint5[22435] = {X 475.9241, Y 30.4499, Z -7.1667, A 0.000, B 0.000, C 0.000 }
gfCNCPoint5[22436] = {X 474.9288, Y 29.2816, Z -7.1667, A 0.000, B 0.000, C 0.000 }
gfCNCPoint5[22437] = {X 474.0999, Y 27.9899, Z -7.1667, A 0.000, B 0.000, C 0.000 }
gfCNCPoint5[22438] = {X 473.4525, Y 26.5984, Z -7.1667, A 0.000, B 0.000, C 0.000 }
gfCNCPoint5[22439] = {X 472.9982, Y 25.1324, Z -7.1667, A 0.000, B 0.000, C 0.000 }
gfCNCPoint5[22440] = {X 472.6860, Y 23.4573, Z -7.1667, A 0.000, B 0.000, C 0.000 }
gfCNCPoint5[22441] = {X 472.5464, Y 21.7591, Z -7.1667, A 0.000, B 0.000, C 0.000 }
gfCNCPoint5[22442] = {X 472.5810, Y 20.0555, Z -7.1667, A 0.000, B 0.000, C 0.000 }
gfCNCPoint5[22443] = {X 472.7892, Y 18.3644, Z -7.1667, A 0.000, B 0.000, C 0.000 }
gfCNCPoint5[22444] = {X 473.1691, Y 16.7033, Z -7.1667, A 0.000, B 0.000, C 0.000 }
gfCNCPoint5[22445] = {X 473.7084, Y 15.1986, Z -7.1667, A 0.000, B 0.000, C 0.000 }
gfCNCPoint5[22446] = {X 474.4469, Y 13.7810, Z -7.1667, A 0.000, B 0.000, C 0.000 }
gfCNCPoint5[22447] = {X 475.3708, Y 12.4767, Z -7.1667, A 0.000, B 0.000, C 0.000 }
gfCNCPoint5[22448] = {X 476.4631, Y 11.3098, Z -7.1667, A 0.000, B 0.000, C 0.000 }
gfCNCPoint5[22449] = {X 477.7037, Y 10.3018, Z -7.1667, A 0.000, B 0.000, C 0.000 }
gfCNCPoint5[22450] = {X 479.0696, Y 9.4715, Z -7.1667, A 0.000, B 0.000, C 0.000 }
gfCNCPoint5[22451] = {X 480.5354, Y 8.8341, Z -7.1667, A 0.000, B 0.000, C 0.000 }
gfCNCPoint5[22452] = {X 482.0742, Y 8.4015, Z -7.1667, A 0.000, B 0.000, C 0.000 }
gfCNCPoint5[22453] = {X 484.1638, Y 8.0764, Z -7.1667, A 0.000, B 0.000, C 0.000 }
gfCNCPoint5[22454] = {X 486.2755, Y 7.9617, Z -7.1667, A 0.000, B 0.000, C 0.000 }
gfCNCPoint5[22455] = {X 486.9686, Y 7.9496, Z -7.1667, A 0.000, B 0.000, C 0.000 }
gfCNCPoint5[22456] = {X 492.3835, Y 7.9496, Z -7.1667, A 0.000, B 0.000, C 0.000 }
gfCNCPoint5[22457] = {X 492.3835, Y 3.9496, Z -7.1667, A 0.000, B 0.000, C 0.000 }
gfCNCPoint5[22458] = {X 492.3835, Y 8.0296, Z -7.1667, A 0.000, B 0.000, C 0.000 }
gfCNCPoint5[22459] = {X 502.2059, Y 8.0296, Z -7.1667, A 0.000, B 0.000, C 0.000 }
gfCNCPoint5[22460] = {X 502.7382, Y 8.0337, Z -7.1667, A 0.000, B 0.000, C 0.000 }
gfCNCPoint5[22461] = {X 503.6547, Y 8.1437, Z -7.1667, A 0.000, B 0.000, C 0.000 }
gfCNCPoint5[22462] = {X 504.5241, Y 8.4539, Z -7.1667, A 0.000, B 0.000, C 0.000 }
gfCNCPoint5[22463] = {X 505.3032, Y 8.9489, Z -7.1667, A 0.000, B 0.000, C 0.000 }
gfCNCPoint5[22464] = {X 505.9533, Y 9.6042, Z -7.1667, A 0.000, B 0.000, C 0.000 }
gfCNCPoint5[22465] = {X 506.4422, Y 10.3871, Z -7.1667, A 0.000, B 0.000, C 0.000 }
gfCNCPoint5[22466] = {X 506.7457, Y 11.2589, Z -7.1667, A 0.000, B 0.000, C 0.000 }
gfCNCPoint5[22467] = {X 506.8485, Y 12.1762, Z -7.1667, A 0.000, B 0.000, C 0.000 }
gfCNCPoint5[22468] = {X 506.8485, Y 12.9782, Z -7.1667, A 0.000, B 0.000, C 0.000 }
gfCNCPoint5[22469] = {X 506.7470, Y 13.8914, Z -7.1667, A 0.000, B 0.000, C 0.000 }
gfCNCPoint5[22470] = {X 506.4475, Y 14.7601, Z -7.1667, A 0.000, B 0.000, C 0.000 }
gfCNCPoint5[22471] = {X 505.9645, Y 15.5418, Z -7.1667, A 0.000, B 0.000, C 0.000 }
gfCNCPoint5[22472] = {X 505.3218, Y 16.1985, Z -7.1667, A 0.000, B 0.000, C 0.000 }
gfCNCPoint5[22473] = {X 505.3221, Y 40.9892, Z -7.1667, A 0.000, B 0.000, C 0.000 }
gfCNCPoint5[22474] = {X 505.3683, Y 41.0269, Z -7.1667, A 0.000, B 0.000, C 0.000 }
gfCNCPoint5[22475] = {X 505.9868, Y 41.6737, Z -7.1667, A 0.000, B 0.000, C 0.000 }
gfCNCPoint5[22476] = {X 506.4527, Y 42.4378, Z -7.1667, A 0.000, B 0.000, C 0.000 }
gfCNCPoint5[22477] = {X 506.7444, Y 43.2838, Z -7.1667, A 0.000, B 0.000, C 0.000 }
gfCNCPoint5[22478] = {X 506.8483, Y 44.1727, Z -7.1667, A 0.000, B 0.000, C 0.000 }
gfCNCPoint5[22479] = {X 506.8485, Y 45.0000, Z -7.1667, A 0.000, B 0.000, C 0.000 }
gfCNCPoint5[22480] = {X 506.7442, Y 45.9257, Z -7.1667, A 0.000, B 0.000, C 0.000 }
gfCNCPoint5[22481] = {X 506.4365, Y 46.8050, Z -7.1667, A 0.000, B 0.000, C 0.000 }
gfCNCPoint5[22482] = {X 505.9409, Y 47.5937, Z -7.1667, A 0.000, B 0.000, C 0.000 }
gfCNCPoint5[22483] = {X 505.2822, Y 48.2524, Z -7.1667, A 0.000, B 0.000, C 0.000 }
gfCNCPoint5[22484] = {X 504.4934, Y 48.7480, Z -7.1667, A 0.000, B 0.000, C 0.000 }
gfCNCPoint5[22485] = {X 503.6142, Y 49.0557, Z -7.1667, A 0.000, B 0.000, C 0.000 }
gfCNCPoint5[22486] = {X 502.6885, Y 49.1600, Z -7.1667, A 0.000, B 0.000, C 0.000 }
gfCNCPoint5[22487] = {X 496.2450, Y 49.1600, Z -7.1667, A 0.000, B 0.000, C 0.000 }
gfCNCPoint5[22488] = {X 495.3239, Y 49.0567, Z -7.1667, A 0.000, B 0.000, C 0.000 }
gfCNCPoint5[22489] = {X 494.4485, Y 48.7521, Z -7.1667, A 0.000, B 0.000, C 0.000 }
gfCNCPoint5[22490] = {X 493.6623, Y 48.2612, Z -7.1667, A 0.000, B 0.000, C 0.000 }
gfCNCPoint5[22491] = {X 493.0043, Y 47.6084, Z -7.1667, A 0.000, B 0.000, C 0.000 }
gfCNCPoint5[22492] = {X 492.5072, Y 46.8261, Z -7.1667, A 0.000, B 0.000, C 0.000 }
gfCNCPoint5[22493] = {X 492.1957, Y 45.9531, Z -7.1667, A 0.000, B 0.000, C 0.000 }
gfCNCPoint5[22494] = {X 492.0852, Y 45.0328, Z -7.1667, A 0.000, B 0.000, C 0.000 }
gfCNCPoint5[22495] = {X 492.0854, Y 44.1516, Z -7.1667, A 0.000, B 0.000, C 0.000 }
gfCNCPoint5[22496] = {X 492.1960, Y 43.2545, Z -7.1667, A 0.000, B 0.000, C 0.000 }
gfCNCPoint5[22497] = {X 492.4976, Y 42.4026, Z -7.1667, A 0.000, B 0.000, C 0.000 }
gfCNCPoint5[22498] = {X 492.9762, Y 41.6358, Z -7.1667, A 0.000, B 0.000, C 0.000 }
gfCNCPoint5[22499] = {X 493.6090, Y 40.9906, Z -7.1667, A 0.000, B 0.000, C 0.000 }
gfCNCPoint5[22500] = {X 493.6090, Y 34.3138, Z -7.1667, A 0.000, B 0.000, C 0.000 }
gfCNCPoint5[22501] = {X 490.6277, Y 34.3138, Z -7.1667, A 0.000, B 0.000, C 0.000 }
gfCNCPoint5[22502] = {X 486.2662, Y 42.8073, Z -7.1667, A 0.000, B 0.000, C 0.000 }
gfCNCPoint5[22503] = {X 486.2944, Y 42.8839, Z -7.1667, A 0.000, B 0.000, C 0.000 }
gfCNCPoint5[22504] = {X 486.4534, Y 43.5191, Z -7.1667, A 0.000, B 0.000, C 0.000 }
gfCNCPoint5[22505] = {X 486.5108, Y 44.1713, Z -7.1667, A 0.000, B 0.000, C 0.000 }
gfCNCPoint5[22506] = {X 486.5110, Y 45.0000, Z -7.1667, A 0.000, B 0.000, C 0.000 }
gfCNCPoint5[22507] = {X 486.4067, Y 45.9257, Z -7.1667, A 0.000, B 0.000, C 0.000 }
gfCNCPoint5[22508] = {X 486.0990, Y 46.8050, Z -7.1667, A 0.000, B 0.000, C 0.000 }
gfCNCPoint5[22509] = {X 485.6034, Y 47.5937, Z -7.1667, A 0.000, B 0.000, C 0.000 }
gfCNCPoint5[22510] = {X 484.9447, Y 48.2524, Z -7.1667, A 0.000, B 0.000, C 0.000 }
gfCNCPoint5[22511] = {X 484.1560, Y 48.7480, Z -7.1667, A 0.000, B 0.000, C 0.000 }
gfCNCPoint5[22512] = {X 483.2767, Y 49.0557, Z -7.1667, A 0.000, B 0.000, C 0.000 }
gfCNCPoint5[22513] = {X 482.3510, Y 49.1600, Z -7.1667, A 0.000, B 0.000, C 0.000 }
gfCNCPoint5[22514] = {X 475.7650, Y 49.1600, Z -7.1667, A 0.000, B 0.000, C 0.000 }
gfCNCPoint5[22515] = {X 474.8393, Y 49.0557, Z -7.1667, A 0.000, B 0.000, C 0.000 }
gfCNCPoint5[22516] = {X 473.9600, Y 48.7480, Z -7.1667, A 0.000, B 0.000, C 0.000 }
gfCNCPoint5[22517] = {X 473.1713, Y 48.2524, Z -7.1667, A 0.000, B 0.000, C 0.000 }
gfCNCPoint5[22518] = {X 472.5126, Y 47.5937, Z -7.1667, A 0.000, B 0.000, C 0.000 }
gfCNCPoint5[22519] = {X 472.0169, Y 46.8050, Z -7.1667, A 0.000, B 0.000, C 0.000 }
gfCNCPoint5[22520] = {X 471.7093, Y 45.9257, Z -7.1667, A 0.000, B 0.000, C 0.000 }
gfCNCPoint5[22521] = {X 471.6050, Y 45.0000, Z -7.1667, A 0.000, B 0.000, C 0.000 }
gfCNCPoint5[22522] = {X 471.6054, Y 44.1516, Z -7.1667, A 0.000, B 0.000, C 0.000 }
gfCNCPoint5[22523] = {X 471.7016, Y 43.3174, Z -7.1667, A 0.000, B 0.000, C 0.000 }
gfCNCPoint5[22524] = {X 471.9634, Y 42.5195, Z -7.1667, A 0.000, B 0.000, C 0.000 }
gfCNCPoint5[22525] = {X 472.3801, Y 41.7905, Z -7.1667, A 0.000, B 0.000, C 0.000 }
gfCNCPoint5[22526] = {X 472.9347, Y 41.1600, Z -7.1667, A 0.000, B 0.000, C 0.000 }
gfCNCPoint5[22527] = {X 473.6046, Y 40.6537, Z -7.1667, A 0.000, B 0.000, C 0.000 }
gfCNCPoint5[22528] = {X 474.3626, Y 40.2923, Z -7.1667, A 0.000, B 0.000, C 0.000 }
gfCNCPoint5[22529] = {X 478.4443, Y 32.3027, Z -7.1667, A 0.000, B 0.000, C 0.000 }
gfCNCPoint5[22530] = {X 477.1666, Y 31.4491, Z -7.1667, A 0.000, B 0.000, C 0.000 }
gfCNCPoint5[22531] = {X 476.0167, Y 30.4300, Z -7.1667, A 0.000, B 0.000, C 0.000 }
gfCNCPoint5[22532] = {X 475.0157, Y 29.2643, Z -7.1667, A 0.000, B 0.000, C 0.000 }
gfCNCPoint5[22533] = {X 474.1822, Y 27.9734, Z -7.1667, A 0.000, B 0.000, C 0.000 }
gfCNCPoint5[22534] = {X 473.5316, Y 26.5813, Z -7.1667, A 0.000, B 0.000, C 0.000 }
gfCNCPoint5[22535] = {X 473.0761, Y 25.1139, Z -7.1667, A 0.000, B 0.000, C 0.000 }
gfCNCPoint5[22536] = {X 472.7653, Y 23.4468, Z -7.1667, A 0.000, B 0.000, C 0.000 }
gfCNCPoint5[22537] = {X 472.6264, Y 21.7567, Z -7.1667, A 0.000, B 0.000, C 0.000 }
gfCNCPoint5[22538] = {X 472.6607, Y 20.0613, Z -7.1667, A 0.000, B 0.000, C 0.000 }
gfCNCPoint5[22539] = {X 472.8680, Y 18.3782, Z -7.1667, A 0.000, B 0.000, C 0.000 }
gfCNCPoint5[22540] = {X 473.2461, Y 16.7251, Z -7.1667, A 0.000, B 0.000, C 0.000 }
gfCNCPoint5[22541] = {X 473.7817, Y 15.2307, Z -7.1667, A 0.000, B 0.000, C 0.000 }
gfCNCPoint5[22542] = {X 474.5151, Y 13.8227, Z -7.1667, A 0.000, B 0.000, C 0.000 }
gfCNCPoint5[22543] = {X 475.4328, Y 12.5273, Z -7.1667, A 0.000, B 0.000, C 0.000 }
gfCNCPoint5[22544] = {X 476.5177, Y 11.3683, Z -7.1667, A 0.000, B 0.000, C 0.000 }
gfCNCPoint5[22545] = {X 477.7498, Y 10.3672, Z -7.1667, A 0.000, B 0.000, C 0.000 }
gfCNCPoint5[22546] = {X 479.1064, Y 9.5425, Z -7.1667, A 0.000, B 0.000, C 0.000 }
gfCNCPoint5[22547] = {X 480.5623, Y 8.9095, Z -7.1667, A 0.000, B 0.000, C 0.000 }
gfCNCPoint5[22548] = {X 482.0906, Y 8.4798, Z -7.1667, A 0.000, B 0.000, C 0.000 }
gfCNCPoint5[22549] = {X 484.1725, Y 8.1559, Z -7.1667, A 0.000, B 0.000, C 0.000 }
gfCNCPoint5[22550] = {X 486.2764, Y 8.0417, Z -7.1667, A 0.000, B 0.000, C 0.000 }
gfCNCPoint5[22551] = {X 486.9693, Y 8.0296, Z -7.1667, A 0.000, B 0.000, C 0.000 }
gfCNCPoint5[22552] = {X 492.3835, Y 8.0296, Z -7.1667, A 0.000, B 0.000, C 0.000 }
gfCNCPoint5[22553] = {X 492.3835, Y 4.0296, Z -7.1667, A 0.000, B 0.000, C 0.000 }
gfCNCPoint5[22554] = {X 492.3835, Y 8.1096, Z -7.1667, A 0.000, B 0.000, C 0.000 }
gfCNCPoint5[22555] = {X 502.2056, Y 8.1096, Z -7.1667, A 0.000, B 0.000, C 0.000 }
gfCNCPoint5[22556] = {X 502.7376, Y 8.1137, Z -7.1667, A 0.000, B 0.000, C 0.000 }
gfCNCPoint5[22557] = {X 503.6364, Y 8.2216, Z -7.1667, A 0.000, B 0.000, C 0.000 }
gfCNCPoint5[22558] = {X 504.4890, Y 8.5258, Z -7.1667, A 0.000, B 0.000, C 0.000 }
gfCNCPoint5[22559] = {X 505.2530, Y 9.0113, Z -7.1667, A 0.000, B 0.000, C 0.000 }
gfCNCPoint5[22560] = {X 505.8906, Y 9.6539, Z -7.1667, A 0.000, B 0.000, C 0.000 }
gfCNCPoint5[22561] = {X 506.3701, Y 10.4217, Z -7.1667, A 0.000, B 0.000, C 0.000 }
gfCNCPoint5[22562] = {X 506.6676, Y 11.2766, Z -7.1667, A 0.000, B 0.000, C 0.000 }
gfCNCPoint5[22563] = {X 506.7685, Y 12.1762, Z -7.1667, A 0.000, B 0.000, C 0.000 }
gfCNCPoint5[22564] = {X 506.7685, Y 12.9782, Z -7.1667, A 0.000, B 0.000, C 0.000 }
gfCNCPoint5[22565] = {X 506.6668, Y 13.8831, Z -7.1667, A 0.000, B 0.000, C 0.000 }
gfCNCPoint5[22566] = {X 506.3670, Y 14.7429, Z -7.1667, A 0.000, B 0.000, C 0.000 }
gfCNCPoint5[22567] = {X 505.8840, Y 15.5148, Z -7.1667, A 0.000, B 0.000, C 0.000 }
gfCNCPoint5[22568] = {X 505.2418, Y 16.1603, Z -7.1667, A 0.000, B 0.000, C 0.000 }
gfCNCPoint5[22569] = {X 505.2421, Y 41.0271, Z -7.1667, A 0.000, B 0.000, C 0.000 }
gfCNCPoint5[22570] = {X 505.3172, Y 41.0885, Z -7.1667, A 0.000, B 0.000, C 0.000 }
gfCNCPoint5[22571] = {X 505.9236, Y 41.7228, Z -7.1667, A 0.000, B 0.000, C 0.000 }
gfCNCPoint5[22572] = {X 506.3804, Y 42.4721, Z -7.1667, A 0.000, B 0.000, C 0.000 }
gfCNCPoint5[22573] = {X 506.6664, Y 43.3018, Z -7.1667, A 0.000, B 0.000, C 0.000 }
gfCNCPoint5[22574] = {X 506.7683, Y 44.1734, Z -7.1667, A 0.000, B 0.000, C 0.000 }
gfCNCPoint5[22575] = {X 506.7685, Y 45.0000, Z -7.1667, A 0.000, B 0.000, C 0.000 }
gfCNCPoint5[22576] = {X 506.6662, Y 45.9079, Z -7.1667, A 0.000, B 0.000, C 0.000 }
gfCNCPoint5[22577] = {X 506.3644, Y 46.7702, Z -7.1667, A 0.000, B 0.000, C 0.000 }
gfCNCPoint5[22578] = {X 505.8784, Y 47.5438, Z -7.1667, A 0.000, B 0.000, C 0.000 }
gfCNCPoint5[22579] = {X 505.2323, Y 48.1899, Z -7.1667, A 0.000, B 0.000, C 0.000 }
gfCNCPoint5[22580] = {X 504.4587, Y 48.6760, Z -7.1667, A 0.000, B 0.000, C 0.000 }
gfCNCPoint5[22581] = {X 503.5964, Y 48.9777, Z -7.1667, A 0.000, B 0.000, C 0.000 }
gfCNCPoint5[22582] = {X 502.6885, Y 49.0800, Z -7.1667, A 0.000, B 0.000, C 0.000 }
gfCNCPoint5[22583] = {X 496.2450, Y 49.0800, Z -7.1667, A 0.000, B 0.000, C 0.000 }
gfCNCPoint5[22584] = {X 495.3416, Y 48.9787, Z -7.1667, A 0.000, B 0.000, C 0.000 }
gfCNCPoint5[22585] = {X 494.4831, Y 48.6799, Z -7.1667, A 0.000, B 0.000, C 0.000 }
gfCNCPoint5[22586] = {X 493.7120, Y 48.1985, Z -7.1667, A 0.000, B 0.000, C 0.000 }
gfCNCPoint5[22587] = {X 493.0667, Y 47.5582, Z -7.1667, A 0.000, B 0.000, C 0.000 }
gfCNCPoint5[22588] = {X 492.5791, Y 46.7909, Z -7.1667, A 0.000, B 0.000, C 0.000 }
gfCNCPoint5[22589] = {X 492.2736, Y 45.9348, Z -7.1667, A 0.000, B 0.000, C 0.000 }
gfCNCPoint5[22590] = {X 492.1652, Y 45.0322, Z -7.1667, A 0.000, B 0.000, C 0.000 }
gfCNCPoint5[22591] = {X 492.1654, Y 44.1527, Z -7.1667, A 0.000, B 0.000, C 0.000 }
gfCNCPoint5[22592] = {X 492.2760, Y 43.2637, Z -7.1667, A 0.000, B 0.000, C 0.000 }
gfCNCPoint5[22593] = {X 492.5779, Y 42.4203, Z -7.1667, A 0.000, B 0.000, C 0.000 }
gfCNCPoint5[22594] = {X 493.0566, Y 41.6631, Z -7.1667, A 0.000, B 0.000, C 0.000 }
gfCNCPoint5[22595] = {X 493.6890, Y 41.0287, Z -7.1667, A 0.000, B 0.000, C 0.000 }
gfCNCPoint5[22596] = {X 493.6890, Y 34.2338, Z -7.1667, A 0.000, B 0.000, C 0.000 }
gfCNCPoint5[22597] = {X 490.5789, Y 34.2338, Z -7.1667, A 0.000, B 0.000, C 0.000 }
gfCNCPoint5[22598] = {X 486.1790, Y 42.8020, Z -7.1667, A 0.000, B 0.000, C 0.000 }
gfCNCPoint5[22599] = {X 486.2189, Y 42.9105, Z -7.1667, A 0.000, B 0.000, C 0.000 }
gfCNCPoint5[22600] = {X 486.3746, Y 43.5329, Z -7.1667, A 0.000, B 0.000, C 0.000 }
gfCNCPoint5[22601] = {X 486.4309, Y 44.1720, Z -7.1667, A 0.000, B 0.000, C 0.000 }
gfCNCPoint5[22602] = {X 486.4310, Y 45.0000, Z -7.1667, A 0.000, B 0.000, C 0.000 }
gfCNCPoint5[22603] = {X 486.3287, Y 45.9079, Z -7.1667, A 0.000, B 0.000, C 0.000 }
gfCNCPoint5[22604] = {X 486.0270, Y 46.7702, Z -7.1667, A 0.000, B 0.000, C 0.000 }
gfCNCPoint5[22605] = {X 485.5409, Y 47.5438, Z -7.1667, A 0.000, B 0.000, C 0.000 }
gfCNCPoint5[22606] = {X 484.8949, Y 48.1899, Z -7.1667, A 0.000, B 0.000, C 0.000 }
gfCNCPoint5[22607] = {X 484.1213, Y 48.6760, Z -7.1667, A 0.000, B 0.000, C 0.000 }
gfCNCPoint5[22608] = {X 483.2589, Y 48.9777, Z -7.1667, A 0.000, B 0.000, C 0.000 }
gfCNCPoint5[22609] = {X 482.3510, Y 49.0800, Z -7.1667, A 0.000, B 0.000, C 0.000 }
gfCNCPoint5[22610] = {X 475.7650, Y 49.0800, Z -7.1667, A 0.000, B 0.000, C 0.000 }
gfCNCPoint5[22611] = {X 474.8571, Y 48.9777, Z -7.1667, A 0.000, B 0.000, C 0.000 }
gfCNCPoint5[22612] = {X 473.9947, Y 48.6760, Z -7.1667, A 0.000, B 0.000, C 0.000 }
gfCNCPoint5[22613] = {X 473.2211, Y 48.1899, Z -7.1667, A 0.000, B 0.000, C 0.000 }
gfCNCPoint5[22614] = {X 472.5751, Y 47.5438, Z -7.1667, A 0.000, B 0.000, C 0.000 }
gfCNCPoint5[22615] = {X 472.0890, Y 46.7702, Z -7.1667, A 0.000, B 0.000, C 0.000 }
gfCNCPoint5[22616] = {X 471.7873, Y 45.9079, Z -7.1667, A 0.000, B 0.000, C 0.000 }
gfCNCPoint5[22617] = {X 471.6850, Y 45.0000, Z -7.1667, A 0.000, B 0.000, C 0.000 }
gfCNCPoint5[22618] = {X 471.6853, Y 44.1527, Z -7.1667, A 0.000, B 0.000, C 0.000 }
gfCNCPoint5[22619] = {X 471.7809, Y 43.3294, Z -7.1667, A 0.000, B 0.000, C 0.000 }
gfCNCPoint5[22620] = {X 472.0408, Y 42.5424, Z -7.1667, A 0.000, B 0.000, C 0.000 }
gfCNCPoint5[22621] = {X 472.4544, Y 41.8242, Z -7.1667, A 0.000, B 0.000, C 0.000 }
gfCNCPoint5[22622] = {X 473.0046, Y 41.2044, Z -7.1667, A 0.000, B 0.000, C 0.000 }
gfCNCPoint5[22623] = {X 473.6687, Y 40.7085, Z -7.1667, A 0.000, B 0.000, C 0.000 }
gfCNCPoint5[22624] = {X 474.4193, Y 40.3571, Z -7.1667, A 0.000, B 0.000, C 0.000 }
gfCNCPoint5[22625] = {X 478.5503, Y 32.2710, Z -7.1667, A 0.000, B 0.000, C 0.000 }
gfCNCPoint5[22626] = {X 477.2659, Y 31.4244, Z -7.1667, A 0.000, B 0.000, C 0.000 }
gfCNCPoint5[22627] = {X 476.1093, Y 30.4100, Z -7.1667, A 0.000, B 0.000, C 0.000 }
gfCNCPoint5[22628] = {X 475.1026, Y 29.2468, Z -7.1667, A 0.000, B 0.000, C 0.000 }
gfCNCPoint5[22629] = {X 474.2644, Y 27.9568, Z -7.1667, A 0.000, B 0.000, C 0.000 }
gfCNCPoint5[22630] = {X 473.6108, Y 26.5642, Z -7.1667, A 0.000, B 0.000, C 0.000 }
gfCNCPoint5[22631] = {X 473.1539, Y 25.0952, Z -7.1667, A 0.000, B 0.000, C 0.000 }
gfCNCPoint5[22632] = {X 472.8446, Y 23.4362, Z -7.1667, A 0.000, B 0.000, C 0.000 }
gfCNCPoint5[22633] = {X 472.7063, Y 21.7543, Z -7.1667, A 0.000, B 0.000, C 0.000 }
gfCNCPoint5[22634] = {X 472.7405, Y 20.0670, Z -7.1667, A 0.000, B 0.000, C 0.000 }
gfCNCPoint5[22635] = {X 472.9468, Y 18.3921, Z -7.1667, A 0.000, B 0.000, C 0.000 }
gfCNCPoint5[22636] = {X 473.3231, Y 16.7469, Z -7.1667, A 0.000, B 0.000, C 0.000 }
gfCNCPoint5[22637] = {X 473.8550, Y 15.2627, Z -7.1667, A 0.000, B 0.000, C 0.000 }
gfCNCPoint5[22638] = {X 474.5834, Y 13.8644, Z -7.1667, A 0.000, B 0.000, C 0.000 }
gfCNCPoint5[22639] = {X 475.4948, Y 12.5778, Z -7.1667, A 0.000, B 0.000, C 0.000 }
gfCNCPoint5[22640] = {X 476.5723, Y 11.4268, Z -7.1667, A 0.000, B 0.000, C 0.000 }
gfCNCPoint5[22641] = {X 477.7959, Y 10.4326, Z -7.1667, A 0.000, B 0.000, C 0.000 }
gfCNCPoint5[22642] = {X 479.1432, Y 9.6135, Z -7.1667, A 0.000, B 0.000, C 0.000 }
gfCNCPoint5[22643] = {X 480.5891, Y 8.9849, Z -7.1667, A 0.000, B 0.000, C 0.000 }
gfCNCPoint5[22644] = {X 482.1069, Y 8.5582, Z -7.1667, A 0.000, B 0.000, C 0.000 }
gfCNCPoint5[22645] = {X 484.1812, Y 8.2354, Z -7.1667, A 0.000, B 0.000, C 0.000 }
gfCNCPoint5[22646] = {X 486.2773, Y 8.1217, Z -7.1667, A 0.000, B 0.000, C 0.000 }
gfCNCPoint5[22647] = {X 486.9700, Y 8.1096, Z -7.1667, A 0.000, B 0.000, C 0.000 }
gfCNCPoint5[22648] = {X 492.3835, Y 8.1096, Z -7.1667, A 0.000, B 0.000, C 0.000 }
gfCNCPoint5[22649] = {X 492.3835, Y 4.1096, Z -7.1667, A 0.000, B 0.000, C 0.000 }
gfCNCPoint5[22650] = {X 492.3835, Y 8.1896, Z -7.1667, A 0.000, B 0.000, C 0.000 }
gfCNCPoint5[22651] = {X 502.2053, Y 8.1896, Z -7.1667, A 0.000, B 0.000, C 0.000 }
gfCNCPoint5[22652] = {X 502.7370, Y 8.1937, Z -7.1667, A 0.000, B 0.000, C 0.000 }
gfCNCPoint5[22653] = {X 503.6181, Y 8.2995, Z -7.1667, A 0.000, B 0.000, C 0.000 }
gfCNCPoint5[22654] = {X 504.4539, Y 8.5977, Z -7.1667, A 0.000, B 0.000, C 0.000 }
gfCNCPoint5[22655] = {X 505.2029, Y 9.0736, Z -7.1667, A 0.000, B 0.000, C 0.000 }
gfCNCPoint5[22656] = {X 505.8279, Y 9.7035, Z -7.1667, A 0.000, B 0.000, C 0.000 }
gfCNCPoint5[22657] = {X 506.2979, Y 10.4562, Z -7.1667, A 0.000, B 0.000, C 0.000 }
gfCNCPoint5[22658] = {X 506.5896, Y 11.2943, Z -7.1667, A 0.000, B 0.000, C 0.000 }
gfCNCPoint5[22659] = {X 506.6885, Y 12.1762, Z -7.1667, A 0.000, B 0.000, C 0.000 }
gfCNCPoint5[22660] = {X 506.6883, Y 13.0192, Z -7.1667, A 0.000, B 0.000, C 0.000 }
gfCNCPoint5[22661] = {X 506.5797, Y 13.9046, Z -7.1667, A 0.000, B 0.000, C 0.000 }
gfCNCPoint5[22662] = {X 506.2776, Y 14.7439, Z -7.1667, A 0.000, B 0.000, C 0.000 }
gfCNCPoint5[22663] = {X 505.7970, Y 15.4954, Z -7.1667, A 0.000, B 0.000, C 0.000 }
gfCNCPoint5[22664] = {X 505.1618, Y 16.1217, Z -7.1667, A 0.000, B 0.000, C 0.000 }
gfCNCPoint5[22665] = {X 505.1621, Y 41.0651, Z -7.1667, A 0.000, B 0.000, C 0.000 }
gfCNCPoint5[22666] = {X 505.3008, Y 41.1796, Z -7.1667, A 0.000, B 0.000, C 0.000 }
gfCNCPoint5[22667] = {X 505.8864, Y 41.8061, Z -7.1667, A 0.000, B 0.000, C 0.000 }
gfCNCPoint5[22668] = {X 506.3251, Y 42.5429, Z -7.1667, A 0.000, B 0.000, C 0.000 }
gfCNCPoint5[22669] = {X 506.5966, Y 43.3563, Z -7.1667, A 0.000, B 0.000, C 0.000 }
gfCNCPoint5[22670] = {X 506.6885, Y 44.2089, Z -7.1667, A 0.000, B 0.000, C 0.000 }
gfCNCPoint5[22671] = {X 506.6885, Y 45.0000, Z -7.1667, A 0.000, B 0.000, C 0.000 }
gfCNCPoint5[22672] = {X 506.5882, Y 45.8901, Z -7.1667, A 0.000, B 0.000, C 0.000 }
gfCNCPoint5[22673] = {X 506.2924, Y 46.7355, Z -7.1667, A 0.000, B 0.000, C 0.000 }
gfCNCPoint5[22674] = {X 505.8158, Y 47.4940, Z -7.1667, A 0.000, B 0.000, C 0.000 }
gfCNCPoint5[22675] = {X 505.1825, Y 48.1273, Z -7.1667, A 0.000, B 0.000, C 0.000 }
gfCNCPoint5[22676] = {X 504.4240, Y 48.6039, Z -7.1667, A 0.000, B 0.000, C 0.000 }
gfCNCPoint5[22677] = {X 503.5786, Y 48.8997, Z -7.1667, A 0.000, B 0.000, C 0.000 }
gfCNCPoint5[22678] = {X 502.6885, Y 49.0000, Z -7.1667, A 0.000, B 0.000, C 0.000 }
gfCNCPoint5[22679] = {X 496.2450, Y 49.0000, Z -7.1667, A 0.000, B 0.000, C 0.000 }
gfCNCPoint5[22680] = {X 495.3549, Y 48.8997, Z -7.1667, A 0.000, B 0.000, C 0.000 }
gfCNCPoint5[22681] = {X 494.5095, Y 48.6039, Z -7.1667, A 0.000, B 0.000, C 0.000 }
gfCNCPoint5[22682] = {X 493.7511, Y 48.1273, Z -7.1667, A 0.000, B 0.000, C 0.000 }
gfCNCPoint5[22683] = {X 493.1177, Y 47.4939, Z -7.1667, A 0.000, B 0.000, C 0.000 }
gfCNCPoint5[22684] = {X 492.6411, Y 46.7355, Z -7.1667, A 0.000, B 0.000, C 0.000 }
gfCNCPoint5[22685] = {X 492.3453, Y 45.8901, Z -7.1667, A 0.000, B 0.000, C 0.000 }
gfCNCPoint5[22686] = {X 492.2450, Y 45.0000, Z -7.1667, A 0.000, B 0.000, C 0.000 }
gfCNCPoint5[22687] = {X 492.2454, Y 44.1538, Z -7.1667, A 0.000, B 0.000, C 0.000 }
gfCNCPoint5[22688] = {X 492.3560, Y 43.2730, Z -7.1667, A 0.000, B 0.000, C 0.000 }
gfCNCPoint5[22689] = {X 492.6582, Y 42.4382, Z -7.1667, A 0.000, B 0.000, C 0.000 }
gfCNCPoint5[22690] = {X 493.1371, Y 41.6907, Z -7.1667, A 0.000, B 0.000, C 0.000 }
gfCNCPoint5[22691] = {X 493.7690, Y 41.0672, Z -7.1667, A 0.000, B 0.000, C 0.000 }
gfCNCPoint5[22692] = {X 493.7690, Y 34.1538, Z -7.1667, A 0.000, B 0.000, C 0.000 }
gfCNCPoint5[22693] = {X 490.7743, Y 34.1538, Z -7.1667, A 0.000, B 0.000, C 0.000 }
gfCNCPoint5[22694] = {X 490.5307, Y 34.1524, Z -7.1667, A 0.000, B 0.000, C 0.000 }
gfCNCPoint5[22695] = {X 486.0918, Y 42.7967, Z -7.1667, A 0.000, B 0.000, C 0.000 }
gfCNCPoint5[22696] = {X 486.1477, Y 42.9499, Z -7.1667, A 0.000, B 0.000, C 0.000 }
gfCNCPoint5[22697] = {X 486.2999, Y 43.5712, Z -7.1667, A 0.000, B 0.000, C 0.000 }
gfCNCPoint5[22698] = {X 486.3510, Y 44.2089, Z -7.1667, A 0.000, B 0.000, C 0.000 }
gfCNCPoint5[22699] = {X 486.3510, Y 45.0000, Z -7.1667, A 0.000, B 0.000, C 0.000 }
gfCNCPoint5[22700] = {X 486.2507, Y 45.8901, Z -7.1667, A 0.000, B 0.000, C 0.000 }
gfCNCPoint5[22701] = {X 485.9549, Y 46.7355, Z -7.1667, A 0.000, B 0.000, C 0.000 }
gfCNCPoint5[22702] = {X 485.4783, Y 47.4940, Z -7.1667, A 0.000, B 0.000, C 0.000 }
gfCNCPoint5[22703] = {X 484.8450, Y 48.1273, Z -7.1667, A 0.000, B 0.000, C 0.000 }
gfCNCPoint5[22704] = {X 484.0866, Y 48.6039, Z -7.1667, A 0.000, B 0.000, C 0.000 }
gfCNCPoint5[22705] = {X 483.2411, Y 48.8997, Z -7.1667, A 0.000, B 0.000, C 0.000 }
gfCNCPoint5[22706] = {X 482.3510, Y 49.0000, Z -7.1667, A 0.000, B 0.000, C 0.000 }
gfCNCPoint5[22707] = {X 475.7650, Y 49.0000, Z -7.1667, A 0.000, B 0.000, C 0.000 }
gfCNCPoint5[22708] = {X 474.8749, Y 48.8997, Z -7.1667, A 0.000, B 0.000, C 0.000 }
gfCNCPoint5[22709] = {X 474.0294, Y 48.6039, Z -7.1667, A 0.000, B 0.000, C 0.000 }
gfCNCPoint5[22710] = {X 473.2710, Y 48.1273, Z -7.1667, A 0.000, B 0.000, C 0.000 }
gfCNCPoint5[22711] = {X 472.6376, Y 47.4940, Z -7.1667, A 0.000, B 0.000, C 0.000 }
gfCNCPoint5[22712] = {X 472.1611, Y 46.7355, Z -7.1667, A 0.000, B 0.000, C 0.000 }
gfCNCPoint5[22713] = {X 471.8652, Y 45.8901, Z -7.1667, A 0.000, B 0.000, C 0.000 }
gfCNCPoint5[22714] = {X 471.7650, Y 45.0000, Z -7.1667, A 0.000, B 0.000, C 0.000 }
gfCNCPoint5[22715] = {X 471.7653, Y 44.1538, Z -7.1667, A 0.000, B 0.000, C 0.000 }
gfCNCPoint5[22716] = {X 471.8601, Y 43.3414, Z -7.1667, A 0.000, B 0.000, C 0.000 }
gfCNCPoint5[22717] = {X 472.1182, Y 42.5654, Z -7.1667, A 0.000, B 0.000, C 0.000 }
gfCNCPoint5[22718] = {X 472.5286, Y 41.8580, Z -7.1667, A 0.000, B 0.000, C 0.000 }
gfCNCPoint5[22719] = {X 473.0744, Y 41.2489, Z -7.1667, A 0.000, B 0.000, C 0.000 }
gfCNCPoint5[22720] = {X 473.7327, Y 40.7635, Z -7.1667, A 0.000, B 0.000, C 0.000 }
gfCNCPoint5[22721] = {X 474.4759, Y 40.4222, Z -7.1667, A 0.000, B 0.000, C 0.000 }
gfCNCPoint5[22722] = {X 478.6566, Y 32.2388, Z -7.1667, A 0.000, B 0.000, C 0.000 }
gfCNCPoint5[22723] = {X 477.3653, Y 31.3994, Z -7.1667, A 0.000, B 0.000, C 0.000 }
gfCNCPoint5[22724] = {X 476.2022, Y 30.3897, Z -7.1667, A 0.000, B 0.000, C 0.000 }
gfCNCPoint5[22725] = {X 475.1895, Y 29.2293, Z -7.1667, A 0.000, B 0.000, C 0.000 }
gfCNCPoint5[22726] = {X 474.3467, Y 27.9401, Z -7.1667, A 0.000, B 0.000, C 0.000 }
gfCNCPoint5[22727] = {X 473.6899, Y 26.5470, Z -7.1667, A 0.000, B 0.000, C 0.000 }
gfCNCPoint5[22728] = {X 473.2317, Y 25.0766, Z -7.1667, A 0.000, B 0.000, C 0.000 }
gfCNCPoint5[22729] = {X 472.9239, Y 23.4256, Z -7.1667, A 0.000, B 0.000, C 0.000 }
gfCNCPoint5[22730] = {X 472.7863, Y 21.7518, Z -7.1667, A 0.000, B 0.000, C 0.000 }
gfCNCPoint5[22731] = {X 472.8203, Y 20.0727, Z -7.1667, A 0.000, B 0.000, C 0.000 }
gfCNCPoint5[22732] = {X 473.0256, Y 18.4059, Z -7.1667, A 0.000, B 0.000, C 0.000 }
gfCNCPoint5[22733] = {X 473.4000, Y 16.7687, Z -7.1667, A 0.000, B 0.000, C 0.000 }
gfCNCPoint5[22734] = {X 473.9283, Y 15.2948, Z -7.1667, A 0.000, B 0.000, C 0.000 }
gfCNCPoint5[22735] = {X 474.6517, Y 13.9061, Z -7.1667, A 0.000, B 0.000, C 0.000 }
gfCNCPoint5[22736] = {X 475.5568, Y 12.6284, Z -7.1667, A 0.000, B 0.000, C 0.000 }
gfCNCPoint5[22737] = {X 476.6268, Y 11.4853, Z -7.1667, A 0.000, B 0.000, C 0.000 }
gfCNCPoint5[22738] = {X 477.8421, Y 10.4979, Z -7.1667, A 0.000, B 0.000, C 0.000 }
gfCNCPoint5[22739] = {X 479.1800, Y 9.6846, Z -7.1667, A 0.000, B 0.000, C 0.000 }
gfCNCPoint5[22740] = {X 480.6159, Y 9.0602, Z -7.1667, A 0.000, B 0.000, C 0.000 }
gfCNCPoint5[22741] = {X 482.1233, Y 8.6365, Z -7.1667, A 0.000, B 0.000, C 0.000 }
gfCNCPoint5[22742] = {X 484.1898, Y 8.3150, Z -7.1667, A 0.000, B 0.000, C 0.000 }
gfCNCPoint5[22743] = {X 486.2782, Y 8.2017, Z -7.1667, A 0.000, B 0.000, C 0.000 }
gfCNCPoint5[22744] = {X 486.9707, Y 8.1896, Z -7.1667, A 0.000, B 0.000, C 0.000 }
gfCNCPoint5[22745] = {X 492.3835, Y 8.1896, Z -7.1667, A 0.000, B 0.000, C 0.000 }
gfCNCPoint5[22746] = {X 492.3835, Y 4.1096, Z -7.1667, A 0.000, B 0.000, C 0.000 }
gfCNCPoint5[22747] = {X 492.3835, Y 4.1096, Z -4.1667, A 0.000, B 0.000, C 0.000 }
gfCNCPoint5[22748] = {X 492.3835, Y 4.1096, Z 11.0000, A 0.000, B 0.000, C 0.000 }
gfCNCPoint5[22749] = {X 533.9634, Y 3.7894, Z 11.0000, A 0.000, B 0.000, C 0.000 }
gfCNCPoint5[22750] = {X 533.9634, Y 3.7894, Z -4.1667, A 0.000, B 0.000, C 0.000 }
gfCNCPoint5[22751] = {X 533.9634, Y 3.7894, Z -7.1667, A 0.000, B 0.000, C 0.000 }
gfCNCPoint5[22752] = {X 533.9633, Y 7.8694, Z -7.1667, A 0.000, B 0.000, C 0.000 }
gfCNCPoint5[22753] = {X 543.7499, Y 7.8696, Z -7.1667, A 0.000, B 0.000, C 0.000 }
gfCNCPoint5[22754] = {X 544.7303, Y 7.9551, Z -7.1667, A 0.000, B 0.000, C 0.000 }
gfCNCPoint5[22755] = {X 545.6660, Y 8.2600, Z -7.1667, A 0.000, B 0.000, C 0.000 }
gfCNCPoint5[22756] = {X 546.5085, Y 8.7686, Z -7.1667, A 0.000, B 0.000, C 0.000 }
gfCNCPoint5[22757] = {X 547.2142, Y 9.4545, Z -7.1667, A 0.000, B 0.000, C 0.000 }
gfCNCPoint5[22758] = {X 547.7466, Y 10.2822, Z -7.1667, A 0.000, B 0.000, C 0.000 }
gfCNCPoint5[22759] = {X 548.0780, Y 11.2088, Z -7.1667, A 0.000, B 0.000, C 0.000 }
gfCNCPoint5[22760] = {X 548.1914, Y 12.1864, Z -7.1667, A 0.000, B 0.000, C 0.000 }
gfCNCPoint5[22761] = {X 548.1912, Y 13.0225, Z -7.1667, A 0.000, B 0.000, C 0.000 }
gfCNCPoint5[22762] = {X 548.0830, Y 13.9400, Z -7.1667, A 0.000, B 0.000, C 0.000 }
gfCNCPoint5[22763] = {X 547.7821, Y 14.8135, Z -7.1667, A 0.000, B 0.000, C 0.000 }
gfCNCPoint5[22764] = {X 547.3024, Y 15.6031, Z -7.1667, A 0.000, B 0.000, C 0.000 }
gfCNCPoint5[22765] = {X 546.6658, Y 16.2726, Z -7.1667, A 0.000, B 0.000, C 0.000 }
gfCNCPoint5[22766] = {X 546.6650, Y 40.9142, Z -7.1667, A 0.000, B 0.000, C 0.000 }
gfCNCPoint5[22767] = {X 546.6867, Y 40.9321, Z -7.1667, A 0.000, B 0.000, C 0.000 }
gfCNCPoint5[22768] = {X 547.3163, Y 41.6020, Z -7.1667, A 0.000, B 0.000, C 0.000 }
gfCNCPoint5[22769] = {X 547.7898, Y 42.3899, Z -7.1667, A 0.000, B 0.000, C 0.000 }
gfCNCPoint5[22770] = {X 548.0860, Y 43.2601, Z -7.1667, A 0.000, B 0.000, C 0.000 }
gfCNCPoint5[22771] = {X 548.1913, Y 44.1733, Z -7.1667, A 0.000, B 0.000, C 0.000 }
gfCNCPoint5[22772] = {X 548.1914, Y 45.0005, Z -7.1667, A 0.000, B 0.000, C 0.000 }
gfCNCPoint5[22773] = {X 548.0780, Y 45.9780, Z -7.1667, A 0.000, B 0.000, C 0.000 }
gfCNCPoint5[22774] = {X 547.7465, Y 46.9046, Z -7.1667, A 0.000, B 0.000, C 0.000 }
gfCNCPoint5[22775] = {X 547.2141, Y 47.7322, Z -7.1667, A 0.000, B 0.000, C 0.000 }
gfCNCPoint5[22776] = {X 546.5084, Y 48.4180, Z -7.1667, A 0.000, B 0.000, C 0.000 }
gfCNCPoint5[22777] = {X 545.6659, Y 48.9266, Z -7.1667, A 0.000, B 0.000, C 0.000 }
gfCNCPoint5[22778] = {X 544.7303, Y 49.2315, Z -7.1667, A 0.000, B 0.000, C 0.000 }
gfCNCPoint5[22779] = {X 543.7499, Y 49.3169, Z -7.1667, A 0.000, B 0.000, C 0.000 }
gfCNCPoint5[22780] = {X 524.0456, Y 49.3173, Z -7.1667, A 0.000, B 0.000, C 0.000 }
gfCNCPoint5[22781] = {X 523.4989, Y 49.9511, Z -7.1667, A 0.000, B 0.000, C 0.000 }
gfCNCPoint5[22782] = {X 522.8438, Y 50.4721, Z -7.1667, A 0.000, B 0.000, C 0.000 }
gfCNCPoint5[22783] = {X 522.1031, Y 50.8620, Z -7.1667, A 0.000, B 0.000, C 0.000 }
gfCNCPoint5[22784] = {X 521.3028, Y 51.1072, Z -7.1667, A 0.000, B 0.000, C 0.000 }
gfCNCPoint5[22785] = {X 520.4708, Y 51.1991, Z -7.1667, A 0.000, B 0.000, C 0.000 }
gfCNCPoint5[22786] = {X 519.7998, Y 51.1991, Z -7.1667, A 0.000, B 0.000, C 0.000 }
gfCNCPoint5[22787] = {X 518.8385, Y 51.0908, Z -7.1667, A 0.000, B 0.000, C 0.000 }
gfCNCPoint5[22788] = {X 517.9254, Y 50.7713, Z -7.1667, A 0.000, B 0.000, C 0.000 }
gfCNCPoint5[22789] = {X 517.1063, Y 50.2566, Z -7.1667, A 0.000, B 0.000, C 0.000 }
gfCNCPoint5[22790] = {X 516.4223, Y 49.5726, Z -7.1667, A 0.000, B 0.000, C 0.000 }
gfCNCPoint5[22791] = {X 515.9076, Y 48.7535, Z -7.1667, A 0.000, B 0.000, C 0.000 }
gfCNCPoint5[22792] = {X 515.5881, Y 47.8404, Z -7.1667, A 0.000, B 0.000, C 0.000 }
gfCNCPoint5[22793] = {X 515.4798, Y 46.8791, Z -7.1667, A 0.000, B 0.000, C 0.000 }
gfCNCPoint5[22794] = {X 515.4798, Y 39.9011, Z -7.1667, A 0.000, B 0.000, C 0.000 }
gfCNCPoint5[22795] = {X 515.5869, Y 38.9451, Z -7.1667, A 0.000, B 0.000, C 0.000 }
gfCNCPoint5[22796] = {X 515.9029, Y 38.0365, Z -7.1667, A 0.000, B 0.000, C 0.000 }
gfCNCPoint5[22797] = {X 516.4121, Y 37.2204, Z -7.1667, A 0.000, B 0.000, C 0.000 }
gfCNCPoint5[22798] = {X 517.0893, Y 36.5372, Z -7.1667, A 0.000, B 0.000, C 0.000 }
gfCNCPoint5[22799] = {X 517.9010, Y 36.0208, Z -7.1667, A 0.000, B 0.000, C 0.000 }
gfCNCPoint5[22800] = {X 518.8067, Y 35.6968, Z -7.1667, A 0.000, B 0.000, C 0.000 }
gfCNCPoint5[22801] = {X 519.7617, Y 35.5813, Z -7.1667, A 0.000, B 0.000, C 0.000 }
